ABB RAPID module: Module1.mod

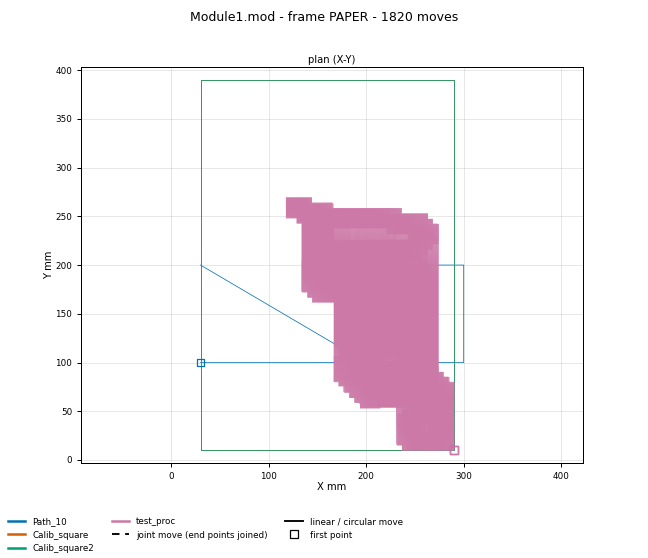
[picture p0: tool path of Module1.mod in frame PAPER, 1820 of 1820 moves have a stored position in this frame; points joined in program order, loops and branches not executed]
MODULE Module1
    CONST robtarget Target_10:=[[30,100,0],[1,0,0,0],[0,0,0,0],[9E+09,9E+09,9E+09,9E+09,9E+09,9E+09]];
    CONST robtarget Target_20:=[[300,100,0],[1,0,0,0],[0,0,0,0],[9E+09,9E+09,9E+09,9E+09,9E+09,9E+09]];
    CONST robtarget Target_30:=[[300,200,0],[1,0,0,0],[0,0,0,0],[9E+09,9E+09,9E+09,9E+09,9E+09,9E+09]];
    CONST robtarget Target_40:=[[200,200,0],[1,0,0,0],[0,0,0,0],[9E+09,9E+09,9E+09,9E+09,9E+09,9E+09]];
    CONST robtarget Target_50:=[[200,100,0],[1,0,0,0],[0,0,0,0],[9E+09,9E+09,9E+09,9E+09,9E+09,9E+09]];
    CONST robtarget Target_60:=[[30,200,0],[1,0,0,0],[0,0,0,0],[9E+09,9E+09,9E+09,9E+09,9E+09,9E+09]];
    CONST robtarget Target_drawing_origin:=[[290,10,-2],[1,0,0,0],[0,0,0,0],[9E+09,9E+09,9E+09,9E+09,9E+09,9E+09]];
!***********************************************************
    !
    ! Module:  Module1
    !
    ! Description:
    !   <Insert description here>
    !
    ! Author: jurdo
    !
    ! Version: 1.0
    !
    !***********************************************************


    !***********************************************************
    !
    ! Procedure main
    !
    !   This is the entry point of your program
    !
    !***********************************************************
    PROC main()

        !Calib_square2;

        test_proc;

    ENDPROC
    PROC Path_10()
        MoveL Target_10,v1000,z0,PencilHolder\WObj:=PAPER;
        MoveL Target_20,v1000,z0,PencilHolder\WObj:=PAPER;
        MoveL Target_30,v1000,z0,PencilHolder\WObj:=PAPER;
        MoveL Target_40,v1000,z0,PencilHolder\WObj:=PAPER;
        MoveL Target_50,v1000,z0,PencilHolder\WObj:=PAPER;
        MoveL Target_60,v1000,z0,PencilHolder\WObj:=PAPER;
    ENDPROC

    PROC Calib_square()
        VAR num width := 380;
        VAR num height := 260;

        MoveJ Offs(Target_drawing_origin,0,0,0),v100,fine,PencilHolder\WObj:=PAPER;

        MoveL Offs(Target_drawing_origin,0,width,0),v100,fine,PencilHolder\WObj:=PAPER;

        MoveL Offs(Target_drawing_origin,-height,width,0),v100,fine,PencilHolder\WObj:=PAPER;

        MoveL Offs(Target_drawing_origin,-height,0,0),v100,fine,PencilHolder\WObj:=PAPER;

        MoveL Offs(Target_drawing_origin,0,0,0),v100,fine,PencilHolder\WObj:=PAPER;

    ENDPROC

    PROC Calib_square2()
    MoveJ Offs(Target_drawing_origin,0,0,0),v100,fine,PencilHolder\WObj:=PAPER;
    MoveL Offs(Target_drawing_origin,0,380,0),v100,fine,PencilHolder\WObj:=PAPER;
    MoveL Offs(Target_drawing_origin,-260,380,0),v100,fine,PencilHolder\WObj:=PAPER;
    MoveL Offs(Target_drawing_origin,-260,0,0),v100,fine,PencilHolder\WObj:=PAPER;
    MoveL Offs(Target_drawing_origin,0,0,0),v100,fine,PencilHolder\WObj:=PAPER;
ENDPROC

! Main procedure
PROC test_proc()


! Draw grey
MoveJ Offs(Target_drawing_origin,0,0,0),v100,fine,PencilHolder\WObj:=PAPER;
MoveL Offs(Target_drawing_origin,0,0,0),v50,fine,PencilHolder\WObj:=PAPER;
MoveL Offs(Target_drawing_origin,0,21,0),v50,fine,PencilHolder\WObj:=PAPER;
MoveL Offs(Target_drawing_origin,0,49,0),v50,fine,PencilHolder\WObj:=PAPER;
MoveL Offs(Target_drawing_origin,0,70,0),v50,fine,PencilHolder\WObj:=PAPER;
MoveL Offs(Target_drawing_origin,-1,0,0),v50,fine,PencilHolder\WObj:=PAPER;
MoveL Offs(Target_drawing_origin,-1,21,0),v50,fine,PencilHolder\WObj:=PAPER;
MoveL Offs(Target_drawing_origin,-1,49,0),v50,fine,PencilHolder\WObj:=PAPER;
MoveL Offs(Target_drawing_origin,-1,70,0),v50,fine,PencilHolder\WObj:=PAPER;
MoveL Offs(Target_drawing_origin,-2,0,0),v50,fine,PencilHolder\WObj:=PAPER;
MoveL Offs(Target_drawing_origin,-2,21,0),v50,fine,PencilHolder\WObj:=PAPER;
MoveL Offs(Target_drawing_origin,-2,49,0),v50,fine,PencilHolder\WObj:=PAPER;
MoveL Offs(Target_drawing_origin,-2,70,0),v50,fine,PencilHolder\WObj:=PAPER;
MoveL Offs(Target_drawing_origin,-3,0,0),v50,fine,PencilHolder\WObj:=PAPER;
MoveL Offs(Target_drawing_origin,-3,21,0),v50,fine,PencilHolder\WObj:=PAPER;
MoveL Offs(Target_drawing_origin,-3,49,0),v50,fine,PencilHolder\WObj:=PAPER;
MoveL Offs(Target_drawing_origin,-3,70,0),v50,fine,PencilHolder\WObj:=PAPER;
MoveL Offs(Target_drawing_origin,-4,0,0),v50,fine,PencilHolder\WObj:=PAPER;
MoveL Offs(Target_drawing_origin,-4,21,0),v50,fine,PencilHolder\WObj:=PAPER;
MoveL Offs(Target_drawing_origin,-4,49,0),v50,fine,PencilHolder\WObj:=PAPER;
MoveL Offs(Target_drawing_origin,-4,70,0),v50,fine,PencilHolder\WObj:=PAPER;
MoveL Offs(Target_drawing_origin,-5,0,0),v50,fine,PencilHolder\WObj:=PAPER;
MoveL Offs(Target_drawing_origin,-5,21,0),v50,fine,PencilHolder\WObj:=PAPER;
MoveL Offs(Target_drawing_origin,-5,44,0),v50,fine,PencilHolder\WObj:=PAPER;
MoveL Offs(Target_drawing_origin,-5,75,0),v50,fine,PencilHolder\WObj:=PAPER;
MoveL Offs(Target_drawing_origin,-6,0,0),v50,fine,PencilHolder\WObj:=PAPER;
MoveL Offs(Target_drawing_origin,-6,21,0),v50,fine,PencilHolder\WObj:=PAPER;
MoveL Offs(Target_drawing_origin,-6,43,0),v50,fine,PencilHolder\WObj:=PAPER;
MoveL Offs(Target_drawing_origin,-6,75,0),v50,fine,PencilHolder\WObj:=PAPER;
MoveL Offs(Target_drawing_origin,-7,0,0),v50,fine,PencilHolder\WObj:=PAPER;
MoveL Offs(Target_drawing_origin,-7,21,0),v50,fine,PencilHolder\WObj:=PAPER;
MoveL Offs(Target_drawing_origin,-7,43,0),v50,fine,PencilHolder\WObj:=PAPER;
MoveL Offs(Target_drawing_origin,-7,75,0),v50,fine,PencilHolder\WObj:=PAPER;
MoveL Offs(Target_drawing_origin,-8,0,0),v50,fine,PencilHolder\WObj:=PAPER;
MoveL Offs(Target_drawing_origin,-8,21,0),v50,fine,PencilHolder\WObj:=PAPER;
MoveL Offs(Target_drawing_origin,-8,43,0),v50,fine,PencilHolder\WObj:=PAPER;
MoveL Offs(Target_drawing_origin,-8,75,0),v50,fine,PencilHolder\WObj:=PAPER;
MoveL Offs(Target_drawing_origin,-9,0,0),v50,fine,PencilHolder\WObj:=PAPER;
MoveL Offs(Target_drawing_origin,-9,21,0),v50,fine,PencilHolder\WObj:=PAPER;
MoveL Offs(Target_drawing_origin,-9,43,0),v50,fine,PencilHolder\WObj:=PAPER;
MoveL Offs(Target_drawing_origin,-9,75,0),v50,fine,PencilHolder\WObj:=PAPER;
MoveL Offs(Target_drawing_origin,-10,0,0),v50,fine,PencilHolder\WObj:=PAPER;
MoveL Offs(Target_drawing_origin,-10,21,0),v50,fine,PencilHolder\WObj:=PAPER;
MoveL Offs(Target_drawing_origin,-10,43,0),v50,fine,PencilHolder\WObj:=PAPER;
MoveL Offs(Target_drawing_origin,-10,75,0),v50,fine,PencilHolder\WObj:=PAPER;
MoveL Offs(Target_drawing_origin,-11,0,0),v50,fine,PencilHolder\WObj:=PAPER;
MoveL Offs(Target_drawing_origin,-11,21,0),v50,fine,PencilHolder\WObj:=PAPER;
MoveL Offs(Target_drawing_origin,-11,38,0),v50,fine,PencilHolder\WObj:=PAPER;
MoveL Offs(Target_drawing_origin,-11,80,0),v50,fine,PencilHolder\WObj:=PAPER;
MoveL Offs(Target_drawing_origin,-12,0,0),v50,fine,PencilHolder\WObj:=PAPER;
MoveL Offs(Target_drawing_origin,-12,21,0),v50,fine,PencilHolder\WObj:=PAPER;
MoveL Offs(Target_drawing_origin,-12,38,0),v50,fine,PencilHolder\WObj:=PAPER;
MoveL Offs(Target_drawing_origin,-12,80,0),v50,fine,PencilHolder\WObj:=PAPER;
MoveL Offs(Target_drawing_origin,-13,0,0),v50,fine,PencilHolder\WObj:=PAPER;
MoveL Offs(Target_drawing_origin,-13,21,0),v50,fine,PencilHolder\WObj:=PAPER;
MoveL Offs(Target_drawing_origin,-13,38,0),v50,fine,PencilHolder\WObj:=PAPER;
MoveL Offs(Target_drawing_origin,-13,80,0),v50,fine,PencilHolder\WObj:=PAPER;
MoveL Offs(Target_drawing_origin,-14,0,0),v50,fine,PencilHolder\WObj:=PAPER;
MoveL Offs(Target_drawing_origin,-14,21,0),v50,fine,PencilHolder\WObj:=PAPER;
MoveL Offs(Target_drawing_origin,-14,38,0),v50,fine,PencilHolder\WObj:=PAPER;
MoveL Offs(Target_drawing_origin,-14,80,0),v50,fine,PencilHolder\WObj:=PAPER;
MoveL Offs(Target_drawing_origin,-15,0,0),v50,fine,PencilHolder\WObj:=PAPER;
MoveL Offs(Target_drawing_origin,-15,21,0),v50,fine,PencilHolder\WObj:=PAPER;
MoveL Offs(Target_drawing_origin,-15,38,0),v50,fine,PencilHolder\WObj:=PAPER;
MoveL Offs(Target_drawing_origin,-15,80,0),v50,fine,PencilHolder\WObj:=PAPER;
MoveL Offs(Target_drawing_origin,-16,0,0),v50,fine,PencilHolder\WObj:=PAPER;
MoveL Offs(Target_drawing_origin,-16,16,0),v50,fine,PencilHolder\WObj:=PAPER;
MoveL Offs(Target_drawing_origin,-16,27,0),v50,fine,PencilHolder\WObj:=PAPER;
MoveL Offs(Target_drawing_origin,-16,86,0),v50,fine,PencilHolder\WObj:=PAPER;
MoveL Offs(Target_drawing_origin,-16,211,0),v50,fine,PencilHolder\WObj:=PAPER;
MoveL Offs(Target_drawing_origin,-16,232,0),v50,fine,PencilHolder\WObj:=PAPER;
MoveL Offs(Target_drawing_origin,-17,0,0),v50,fine,PencilHolder\WObj:=PAPER;
MoveL Offs(Target_drawing_origin,-17,15,0),v50,fine,PencilHolder\WObj:=PAPER;
MoveL Offs(Target_drawing_origin,-17,27,0),v50,fine,PencilHolder\WObj:=PAPER;
MoveL Offs(Target_drawing_origin,-17,86,0),v50,fine,PencilHolder\WObj:=PAPER;
MoveL Offs(Target_drawing_origin,-17,211,0),v50,fine,PencilHolder\WObj:=PAPER;
MoveL Offs(Target_drawing_origin,-17,232,0),v50,fine,PencilHolder\WObj:=PAPER;
MoveL Offs(Target_drawing_origin,-18,0,0),v50,fine,PencilHolder\WObj:=PAPER;
MoveL Offs(Target_drawing_origin,-18,15,0),v50,fine,PencilHolder\WObj:=PAPER;
MoveL Offs(Target_drawing_origin,-18,27,0),v50,fine,PencilHolder\WObj:=PAPER;
MoveL Offs(Target_drawing_origin,-18,86,0),v50,fine,PencilHolder\WObj:=PAPER;
MoveL Offs(Target_drawing_origin,-18,211,0),v50,fine,PencilHolder\WObj:=PAPER;
MoveL Offs(Target_drawing_origin,-18,232,0),v50,fine,PencilHolder\WObj:=PAPER;
MoveL Offs(Target_drawing_origin,-19,0,0),v50,fine,PencilHolder\WObj:=PAPER;
MoveL Offs(Target_drawing_origin,-19,15,0),v50,fine,PencilHolder\WObj:=PAPER;
MoveL Offs(Target_drawing_origin,-19,27,0),v50,fine,PencilHolder\WObj:=PAPER;
MoveL Offs(Target_drawing_origin,-19,86,0),v50,fine,PencilHolder\WObj:=PAPER;
MoveL Offs(Target_drawing_origin,-19,211,0),v50,fine,PencilHolder\WObj:=PAPER;
MoveL Offs(Target_drawing_origin,-19,232,0),v50,fine,PencilHolder\WObj:=PAPER;
MoveL Offs(Target_drawing_origin,-20,0,0),v50,fine,PencilHolder\WObj:=PAPER;
MoveL Offs(Target_drawing_origin,-20,15,0),v50,fine,PencilHolder\WObj:=PAPER;
MoveL Offs(Target_drawing_origin,-20,27,0),v50,fine,PencilHolder\WObj:=PAPER;
MoveL Offs(Target_drawing_origin,-20,86,0),v50,fine,PencilHolder\WObj:=PAPER;
MoveL Offs(Target_drawing_origin,-20,211,0),v50,fine,PencilHolder\WObj:=PAPER;
MoveL Offs(Target_drawing_origin,-20,232,0),v50,fine,PencilHolder\WObj:=PAPER;
MoveL Offs(Target_drawing_origin,-21,0,0),v50,fine,PencilHolder\WObj:=PAPER;
MoveL Offs(Target_drawing_origin,-21,15,0),v50,fine,PencilHolder\WObj:=PAPER;
MoveL Offs(Target_drawing_origin,-21,27,0),v50,fine,PencilHolder\WObj:=PAPER;
MoveL Offs(Target_drawing_origin,-21,86,0),v50,fine,PencilHolder\WObj:=PAPER;
MoveL Offs(Target_drawing_origin,-21,211,0),v50,fine,PencilHolder\WObj:=PAPER;
MoveL Offs(Target_drawing_origin,-21,232,0),v50,fine,PencilHolder\WObj:=PAPER;
MoveL Offs(Target_drawing_origin,-22,0,0),v50,fine,PencilHolder\WObj:=PAPER;
MoveL Offs(Target_drawing_origin,-22,15,0),v50,fine,PencilHolder\WObj:=PAPER;
MoveL Offs(Target_drawing_origin,-22,27,0),v50,fine,PencilHolder\WObj:=PAPER;
MoveL Offs(Target_drawing_origin,-22,91,0),v50,fine,PencilHolder\WObj:=PAPER;
MoveL Offs(Target_drawing_origin,-22,206,0),v50,fine,PencilHolder\WObj:=PAPER;
MoveL Offs(Target_drawing_origin,-22,237,0),v50,fine,PencilHolder\WObj:=PAPER;
MoveL Offs(Target_drawing_origin,-23,0,0),v50,fine,PencilHolder\WObj:=PAPER;
MoveL Offs(Target_drawing_origin,-23,15,0),v50,fine,PencilHolder\WObj:=PAPER;
MoveL Offs(Target_drawing_origin,-23,27,0),v50,fine,PencilHolder\WObj:=PAPER;
MoveL Offs(Target_drawing_origin,-23,91,0),v50,fine,PencilHolder\WObj:=PAPER;
MoveL Offs(Target_drawing_origin,-23,206,0),v50,fine,PencilHolder\WObj:=PAPER;
MoveL Offs(Target_drawing_origin,-23,237,0),v50,fine,PencilHolder\WObj:=PAPER;
MoveL Offs(Target_drawing_origin,-24,0,0),v50,fine,PencilHolder\WObj:=PAPER;
MoveL Offs(Target_drawing_origin,-24,15,0),v50,fine,PencilHolder\WObj:=PAPER;
MoveL Offs(Target_drawing_origin,-24,27,0),v50,fine,PencilHolder\WObj:=PAPER;
MoveL Offs(Target_drawing_origin,-24,91,0),v50,fine,PencilHolder\WObj:=PAPER;
MoveL Offs(Target_drawing_origin,-24,206,0),v50,fine,PencilHolder\WObj:=PAPER;
MoveL Offs(Target_drawing_origin,-24,237,0),v50,fine,PencilHolder\WObj:=PAPER;
MoveL Offs(Target_drawing_origin,-25,0,0),v50,fine,PencilHolder\WObj:=PAPER;
MoveL Offs(Target_drawing_origin,-25,15,0),v50,fine,PencilHolder\WObj:=PAPER;
MoveL Offs(Target_drawing_origin,-25,27,0),v50,fine,PencilHolder\WObj:=PAPER;
MoveL Offs(Target_drawing_origin,-25,91,0),v50,fine,PencilHolder\WObj:=PAPER;
MoveL Offs(Target_drawing_origin,-25,206,0),v50,fine,PencilHolder\WObj:=PAPER;
MoveL Offs(Target_drawing_origin,-25,237,0),v50,fine,PencilHolder\WObj:=PAPER;
MoveL Offs(Target_drawing_origin,-26,0,0),v50,fine,PencilHolder\WObj:=PAPER;
MoveL Offs(Target_drawing_origin,-26,15,0),v50,fine,PencilHolder\WObj:=PAPER;
MoveL Offs(Target_drawing_origin,-26,27,0),v50,fine,PencilHolder\WObj:=PAPER;
MoveL Offs(Target_drawing_origin,-26,91,0),v50,fine,PencilHolder\WObj:=PAPER;
MoveL Offs(Target_drawing_origin,-26,206,0),v50,fine,PencilHolder\WObj:=PAPER;
MoveL Offs(Target_drawing_origin,-26,237,0),v50,fine,PencilHolder\WObj:=PAPER;
MoveL Offs(Target_drawing_origin,-27,0,0),v50,fine,PencilHolder\WObj:=PAPER;
MoveL Offs(Target_drawing_origin,-27,91,0),v50,fine,PencilHolder\WObj:=PAPER;
MoveL Offs(Target_drawing_origin,-27,131,0),v50,fine,PencilHolder\WObj:=PAPER;
MoveL Offs(Target_drawing_origin,-27,156,0),v50,fine,PencilHolder\WObj:=PAPER;
MoveL Offs(Target_drawing_origin,-27,200,0),v50,fine,PencilHolder\WObj:=PAPER;
MoveL Offs(Target_drawing_origin,-27,243,0),v50,fine,PencilHolder\WObj:=PAPER;
MoveL Offs(Target_drawing_origin,-28,0,0),v50,fine,PencilHolder\WObj:=PAPER;
MoveL Offs(Target_drawing_origin,-28,91,0),v50,fine,PencilHolder\WObj:=PAPER;
MoveL Offs(Target_drawing_origin,-28,131,0),v50,fine,PencilHolder\WObj:=PAPER;
MoveL Offs(Target_drawing_origin,-28,156,0),v50,fine,PencilHolder\WObj:=PAPER;
MoveL Offs(Target_drawing_origin,-28,200,0),v50,fine,PencilHolder\WObj:=PAPER;
MoveL Offs(Target_drawing_origin,-28,243,0),v50,fine,PencilHolder\WObj:=PAPER;
MoveL Offs(Target_drawing_origin,-29,0,0),v50,fine,PencilHolder\WObj:=PAPER;
MoveL Offs(Target_drawing_origin,-29,91,0),v50,fine,PencilHolder\WObj:=PAPER;
MoveL Offs(Target_drawing_origin,-29,131,0),v50,fine,PencilHolder\WObj:=PAPER;
MoveL Offs(Target_drawing_origin,-29,156,0),v50,fine,PencilHolder\WObj:=PAPER;
MoveL Offs(Target_drawing_origin,-29,200,0),v50,fine,PencilHolder\WObj:=PAPER;
MoveL Offs(Target_drawing_origin,-29,243,0),v50,fine,PencilHolder\WObj:=PAPER;
MoveL Offs(Target_drawing_origin,-30,0,0),v50,fine,PencilHolder\WObj:=PAPER;
MoveL Offs(Target_drawing_origin,-30,91,0),v50,fine,PencilHolder\WObj:=PAPER;
MoveL Offs(Target_drawing_origin,-30,131,0),v50,fine,PencilHolder\WObj:=PAPER;
MoveL Offs(Target_drawing_origin,-30,156,0),v50,fine,PencilHolder\WObj:=PAPER;
MoveL Offs(Target_drawing_origin,-30,200,0),v50,fine,PencilHolder\WObj:=PAPER;
MoveL Offs(Target_drawing_origin,-30,243,0),v50,fine,PencilHolder\WObj:=PAPER;
MoveL Offs(Target_drawing_origin,-31,0,0),v50,fine,PencilHolder\WObj:=PAPER;
MoveL Offs(Target_drawing_origin,-31,91,0),v50,fine,PencilHolder\WObj:=PAPER;
MoveL Offs(Target_drawing_origin,-31,131,0),v50,fine,PencilHolder\WObj:=PAPER;
MoveL Offs(Target_drawing_origin,-31,156,0),v50,fine,PencilHolder\WObj:=PAPER;
MoveL Offs(Target_drawing_origin,-31,200,0),v50,fine,PencilHolder\WObj:=PAPER;
MoveL Offs(Target_drawing_origin,-31,243,0),v50,fine,PencilHolder\WObj:=PAPER;
MoveL Offs(Target_drawing_origin,-32,0,0),v50,fine,PencilHolder\WObj:=PAPER;
MoveL Offs(Target_drawing_origin,-32,91,0),v50,fine,PencilHolder\WObj:=PAPER;
MoveL Offs(Target_drawing_origin,-32,125,0),v50,fine,PencilHolder\WObj:=PAPER;
MoveL Offs(Target_drawing_origin,-32,161,0),v50,fine,PencilHolder\WObj:=PAPER;
MoveL Offs(Target_drawing_origin,-32,195,0),v50,fine,PencilHolder\WObj:=PAPER;
MoveL Offs(Target_drawing_origin,-32,243,0),v50,fine,PencilHolder\WObj:=PAPER;
MoveL Offs(Target_drawing_origin,-33,0,0),v50,fine,PencilHolder\WObj:=PAPER;
MoveL Offs(Target_drawing_origin,-33,53,0),v50,fine,PencilHolder\WObj:=PAPER;
MoveL Offs(Target_drawing_origin,-33,59,0),v50,fine,PencilHolder\WObj:=PAPER;
MoveL Offs(Target_drawing_origin,-33,91,0),v50,fine,PencilHolder\WObj:=PAPER;
MoveL Offs(Target_drawing_origin,-33,124,0),v50,fine,PencilHolder\WObj:=PAPER;
MoveL Offs(Target_drawing_origin,-33,162,0),v50,fine,PencilHolder\WObj:=PAPER;
MoveL Offs(Target_drawing_origin,-33,195,0),v50,fine,PencilHolder\WObj:=PAPER;
MoveL Offs(Target_drawing_origin,-33,243,0),v50,fine,PencilHolder\WObj:=PAPER;
MoveL Offs(Target_drawing_origin,-34,0,0),v50,fine,PencilHolder\WObj:=PAPER;
MoveL Offs(Target_drawing_origin,-34,53,0),v50,fine,PencilHolder\WObj:=PAPER;
MoveL Offs(Target_drawing_origin,-34,59,0),v50,fine,PencilHolder\WObj:=PAPER;
MoveL Offs(Target_drawing_origin,-34,91,0),v50,fine,PencilHolder\WObj:=PAPER;
MoveL Offs(Target_drawing_origin,-34,124,0),v50,fine,PencilHolder\WObj:=PAPER;
MoveL Offs(Target_drawing_origin,-34,162,0),v50,fine,PencilHolder\WObj:=PAPER;
MoveL Offs(Target_drawing_origin,-34,195,0),v50,fine,PencilHolder\WObj:=PAPER;
MoveL Offs(Target_drawing_origin,-34,243,0),v50,fine,PencilHolder\WObj:=PAPER;
MoveL Offs(Target_drawing_origin,-35,0,0),v50,fine,PencilHolder\WObj:=PAPER;
MoveL Offs(Target_drawing_origin,-35,53,0),v50,fine,PencilHolder\WObj:=PAPER;
MoveL Offs(Target_drawing_origin,-35,59,0),v50,fine,PencilHolder\WObj:=PAPER;
MoveL Offs(Target_drawing_origin,-35,91,0),v50,fine,PencilHolder\WObj:=PAPER;
MoveL Offs(Target_drawing_origin,-35,124,0),v50,fine,PencilHolder\WObj:=PAPER;
MoveL Offs(Target_drawing_origin,-35,162,0),v50,fine,PencilHolder\WObj:=PAPER;
MoveL Offs(Target_drawing_origin,-35,195,0),v50,fine,PencilHolder\WObj:=PAPER;
MoveL Offs(Target_drawing_origin,-35,243,0),v50,fine,PencilHolder\WObj:=PAPER;
MoveL Offs(Target_drawing_origin,-36,0,0),v50,fine,PencilHolder\WObj:=PAPER;
MoveL Offs(Target_drawing_origin,-36,53,0),v50,fine,PencilHolder\WObj:=PAPER;
MoveL Offs(Target_drawing_origin,-36,59,0),v50,fine,PencilHolder\WObj:=PAPER;
MoveL Offs(Target_drawing_origin,-36,91,0),v50,fine,PencilHolder\WObj:=PAPER;
MoveL Offs(Target_drawing_origin,-36,124,0),v50,fine,PencilHolder\WObj:=PAPER;
MoveL Offs(Target_drawing_origin,-36,162,0),v50,fine,PencilHolder\WObj:=PAPER;
MoveL Offs(Target_drawing_origin,-36,195,0),v50,fine,PencilHolder\WObj:=PAPER;
MoveL Offs(Target_drawing_origin,-36,243,0),v50,fine,PencilHolder\WObj:=PAPER;
MoveL Offs(Target_drawing_origin,-37,0,0),v50,fine,PencilHolder\WObj:=PAPER;
MoveL Offs(Target_drawing_origin,-37,53,0),v50,fine,PencilHolder\WObj:=PAPER;
MoveL Offs(Target_drawing_origin,-37,59,0),v50,fine,PencilHolder\WObj:=PAPER;
MoveL Offs(Target_drawing_origin,-37,91,0),v50,fine,PencilHolder\WObj:=PAPER;
MoveL Offs(Target_drawing_origin,-37,124,0),v50,fine,PencilHolder\WObj:=PAPER;
MoveL Offs(Target_drawing_origin,-37,162,0),v50,fine,PencilHolder\WObj:=PAPER;
MoveL Offs(Target_drawing_origin,-37,195,0),v50,fine,PencilHolder\WObj:=PAPER;
MoveL Offs(Target_drawing_origin,-37,243,0),v50,fine,PencilHolder\WObj:=PAPER;
MoveL Offs(Target_drawing_origin,-38,0,0),v50,fine,PencilHolder\WObj:=PAPER;
MoveL Offs(Target_drawing_origin,-38,48,0),v50,fine,PencilHolder\WObj:=PAPER;
MoveL Offs(Target_drawing_origin,-38,59,0),v50,fine,PencilHolder\WObj:=PAPER;
MoveL Offs(Target_drawing_origin,-38,91,0),v50,fine,PencilHolder\WObj:=PAPER;
MoveL Offs(Target_drawing_origin,-38,114,0),v50,fine,PencilHolder\WObj:=PAPER;
MoveL Offs(Target_drawing_origin,-38,167,0),v50,fine,PencilHolder\WObj:=PAPER;
MoveL Offs(Target_drawing_origin,-38,195,0),v50,fine,PencilHolder\WObj:=PAPER;
MoveL Offs(Target_drawing_origin,-38,243,0),v50,fine,PencilHolder\WObj:=PAPER;
MoveL Offs(Target_drawing_origin,-39,0,0),v50,fine,PencilHolder\WObj:=PAPER;
MoveL Offs(Target_drawing_origin,-39,48,0),v50,fine,PencilHolder\WObj:=PAPER;
MoveL Offs(Target_drawing_origin,-39,59,0),v50,fine,PencilHolder\WObj:=PAPER;
MoveL Offs(Target_drawing_origin,-39,91,0),v50,fine,PencilHolder\WObj:=PAPER;
MoveL Offs(Target_drawing_origin,-39,114,0),v50,fine,PencilHolder\WObj:=PAPER;
MoveL Offs(Target_drawing_origin,-39,167,0),v50,fine,PencilHolder\WObj:=PAPER;
MoveL Offs(Target_drawing_origin,-39,195,0),v50,fine,PencilHolder\WObj:=PAPER;
MoveL Offs(Target_drawing_origin,-39,243,0),v50,fine,PencilHolder\WObj:=PAPER;
MoveL Offs(Target_drawing_origin,-40,0,0),v50,fine,PencilHolder\WObj:=PAPER;
MoveL Offs(Target_drawing_origin,-40,48,0),v50,fine,PencilHolder\WObj:=PAPER;
MoveL Offs(Target_drawing_origin,-40,59,0),v50,fine,PencilHolder\WObj:=PAPER;
MoveL Offs(Target_drawing_origin,-40,91,0),v50,fine,PencilHolder\WObj:=PAPER;
MoveL Offs(Target_drawing_origin,-40,114,0),v50,fine,PencilHolder\WObj:=PAPER;
MoveL Offs(Target_drawing_origin,-40,167,0),v50,fine,PencilHolder\WObj:=PAPER;
MoveL Offs(Target_drawing_origin,-40,195,0),v50,fine,PencilHolder\WObj:=PAPER;
MoveL Offs(Target_drawing_origin,-40,243,0),v50,fine,PencilHolder\WObj:=PAPER;
MoveL Offs(Target_drawing_origin,-41,0,0),v50,fine,PencilHolder\WObj:=PAPER;
MoveL Offs(Target_drawing_origin,-41,48,0),v50,fine,PencilHolder\WObj:=PAPER;
MoveL Offs(Target_drawing_origin,-41,59,0),v50,fine,PencilHolder\WObj:=PAPER;
MoveL Offs(Target_drawing_origin,-41,91,0),v50,fine,PencilHolder\WObj:=PAPER;
MoveL Offs(Target_drawing_origin,-41,114,0),v50,fine,PencilHolder\WObj:=PAPER;
MoveL Offs(Target_drawing_origin,-41,167,0),v50,fine,PencilHolder\WObj:=PAPER;
MoveL Offs(Target_drawing_origin,-41,195,0),v50,fine,PencilHolder\WObj:=PAPER;
MoveL Offs(Target_drawing_origin,-41,243,0),v50,fine,PencilHolder\WObj:=PAPER;
MoveL Offs(Target_drawing_origin,-42,0,0),v50,fine,PencilHolder\WObj:=PAPER;
MoveL Offs(Target_drawing_origin,-42,48,0),v50,fine,PencilHolder\WObj:=PAPER;
MoveL Offs(Target_drawing_origin,-42,59,0),v50,fine,PencilHolder\WObj:=PAPER;
MoveL Offs(Target_drawing_origin,-42,91,0),v50,fine,PencilHolder\WObj:=PAPER;
MoveL Offs(Target_drawing_origin,-42,114,0),v50,fine,PencilHolder\WObj:=PAPER;
MoveL Offs(Target_drawing_origin,-42,167,0),v50,fine,PencilHolder\WObj:=PAPER;
MoveL Offs(Target_drawing_origin,-42,195,0),v50,fine,PencilHolder\WObj:=PAPER;
MoveL Offs(Target_drawing_origin,-42,243,0),v50,fine,PencilHolder\WObj:=PAPER;
MoveL Offs(Target_drawing_origin,-43,0,0),v50,fine,PencilHolder\WObj:=PAPER;
MoveL Offs(Target_drawing_origin,-43,43,0),v50,fine,PencilHolder\WObj:=PAPER;
MoveL Offs(Target_drawing_origin,-43,59,0),v50,fine,PencilHolder\WObj:=PAPER;
MoveL Offs(Target_drawing_origin,-43,91,0),v50,fine,PencilHolder\WObj:=PAPER;
MoveL Offs(Target_drawing_origin,-43,108,0),v50,fine,PencilHolder\WObj:=PAPER;
MoveL Offs(Target_drawing_origin,-43,172,0),v50,fine,PencilHolder\WObj:=PAPER;
MoveL Offs(Target_drawing_origin,-43,190,0),v50,fine,PencilHolder\WObj:=PAPER;
MoveL Offs(Target_drawing_origin,-43,243,0),v50,fine,PencilHolder\WObj:=PAPER;
MoveL Offs(Target_drawing_origin,-44,0,0),v50,fine,PencilHolder\WObj:=PAPER;
MoveL Offs(Target_drawing_origin,-44,42,0),v50,fine,PencilHolder\WObj:=PAPER;
MoveL Offs(Target_drawing_origin,-44,59,0),v50,fine,PencilHolder\WObj:=PAPER;
MoveL Offs(Target_drawing_origin,-44,91,0),v50,fine,PencilHolder\WObj:=PAPER;
MoveL Offs(Target_drawing_origin,-44,108,0),v50,fine,PencilHolder\WObj:=PAPER;
MoveL Offs(Target_drawing_origin,-44,172,0),v50,fine,PencilHolder\WObj:=PAPER;
MoveL Offs(Target_drawing_origin,-44,189,0),v50,fine,PencilHolder\WObj:=PAPER;
MoveL Offs(Target_drawing_origin,-44,243,0),v50,fine,PencilHolder\WObj:=PAPER;
MoveL Offs(Target_drawing_origin,-45,0,0),v50,fine,PencilHolder\WObj:=PAPER;
MoveL Offs(Target_drawing_origin,-45,42,0),v50,fine,PencilHolder\WObj:=PAPER;
MoveL Offs(Target_drawing_origin,-45,59,0),v50,fine,PencilHolder\WObj:=PAPER;
MoveL Offs(Target_drawing_origin,-45,91,0),v50,fine,PencilHolder\WObj:=PAPER;
MoveL Offs(Target_drawing_origin,-45,108,0),v50,fine,PencilHolder\WObj:=PAPER;
MoveL Offs(Target_drawing_origin,-45,172,0),v50,fine,PencilHolder\WObj:=PAPER;
MoveL Offs(Target_drawing_origin,-45,189,0),v50,fine,PencilHolder\WObj:=PAPER;
MoveL Offs(Target_drawing_origin,-45,243,0),v50,fine,PencilHolder\WObj:=PAPER;
MoveL Offs(Target_drawing_origin,-46,0,0),v50,fine,PencilHolder\WObj:=PAPER;
MoveL Offs(Target_drawing_origin,-46,42,0),v50,fine,PencilHolder\WObj:=PAPER;
MoveL Offs(Target_drawing_origin,-46,59,0),v50,fine,PencilHolder\WObj:=PAPER;
MoveL Offs(Target_drawing_origin,-46,91,0),v50,fine,PencilHolder\WObj:=PAPER;
MoveL Offs(Target_drawing_origin,-46,108,0),v50,fine,PencilHolder\WObj:=PAPER;
MoveL Offs(Target_drawing_origin,-46,172,0),v50,fine,PencilHolder\WObj:=PAPER;
MoveL Offs(Target_drawing_origin,-46,189,0),v50,fine,PencilHolder\WObj:=PAPER;
MoveL Offs(Target_drawing_origin,-46,243,0),v50,fine,PencilHolder\WObj:=PAPER;
MoveL Offs(Target_drawing_origin,-47,0,0),v50,fine,PencilHolder\WObj:=PAPER;
MoveL Offs(Target_drawing_origin,-47,42,0),v50,fine,PencilHolder\WObj:=PAPER;
MoveL Offs(Target_drawing_origin,-47,59,0),v50,fine,PencilHolder\WObj:=PAPER;
MoveL Offs(Target_drawing_origin,-47,91,0),v50,fine,PencilHolder\WObj:=PAPER;
MoveL Offs(Target_drawing_origin,-47,108,0),v50,fine,PencilHolder\WObj:=PAPER;
MoveL Offs(Target_drawing_origin,-47,172,0),v50,fine,PencilHolder\WObj:=PAPER;
MoveL Offs(Target_drawing_origin,-47,189,0),v50,fine,PencilHolder\WObj:=PAPER;
MoveL Offs(Target_drawing_origin,-47,243,0),v50,fine,PencilHolder\WObj:=PAPER;
MoveL Offs(Target_drawing_origin,-48,0,0),v50,fine,PencilHolder\WObj:=PAPER;
MoveL Offs(Target_drawing_origin,-48,42,0),v50,fine,PencilHolder\WObj:=PAPER;
MoveL Offs(Target_drawing_origin,-48,59,0),v50,fine,PencilHolder\WObj:=PAPER;
MoveL Offs(Target_drawing_origin,-48,91,0),v50,fine,PencilHolder\WObj:=PAPER;
MoveL Offs(Target_drawing_origin,-48,108,0),v50,fine,PencilHolder\WObj:=PAPER;
MoveL Offs(Target_drawing_origin,-48,172,0),v50,fine,PencilHolder\WObj:=PAPER;
MoveL Offs(Target_drawing_origin,-48,189,0),v50,fine,PencilHolder\WObj:=PAPER;
MoveL Offs(Target_drawing_origin,-48,243,0),v50,fine,PencilHolder\WObj:=PAPER;
MoveL Offs(Target_drawing_origin,-49,0,0),v50,fine,PencilHolder\WObj:=PAPER;
MoveL Offs(Target_drawing_origin,-49,42,0),v50,fine,PencilHolder\WObj:=PAPER;
MoveL Offs(Target_drawing_origin,-49,59,0),v50,fine,PencilHolder\WObj:=PAPER;
MoveL Offs(Target_drawing_origin,-49,91,0),v50,fine,PencilHolder\WObj:=PAPER;
MoveL Offs(Target_drawing_origin,-49,103,0),v50,fine,PencilHolder\WObj:=PAPER;
MoveL Offs(Target_drawing_origin,-49,172,0),v50,fine,PencilHolder\WObj:=PAPER;
MoveL Offs(Target_drawing_origin,-49,189,0),v50,fine,PencilHolder\WObj:=PAPER;
MoveL Offs(Target_drawing_origin,-49,216,0),v50,fine,PencilHolder\WObj:=PAPER;
MoveL Offs(Target_drawing_origin,-49,222,0),v50,fine,PencilHolder\WObj:=PAPER;
MoveL Offs(Target_drawing_origin,-49,243,0),v50,fine,PencilHolder\WObj:=PAPER;
MoveL Offs(Target_drawing_origin,-50,0,0),v50,fine,PencilHolder\WObj:=PAPER;
MoveL Offs(Target_drawing_origin,-50,42,0),v50,fine,PencilHolder\WObj:=PAPER;
MoveL Offs(Target_drawing_origin,-50,59,0),v50,fine,PencilHolder\WObj:=PAPER;
MoveL Offs(Target_drawing_origin,-50,91,0),v50,fine,PencilHolder\WObj:=PAPER;
MoveL Offs(Target_drawing_origin,-50,103,0),v50,fine,PencilHolder\WObj:=PAPER;
MoveL Offs(Target_drawing_origin,-50,172,0),v50,fine,PencilHolder\WObj:=PAPER;
MoveL Offs(Target_drawing_origin,-50,189,0),v50,fine,PencilHolder\WObj:=PAPER;
MoveL Offs(Target_drawing_origin,-50,216,0),v50,fine,PencilHolder\WObj:=PAPER;
MoveL Offs(Target_drawing_origin,-50,222,0),v50,fine,PencilHolder\WObj:=PAPER;
MoveL Offs(Target_drawing_origin,-50,243,0),v50,fine,PencilHolder\WObj:=PAPER;
MoveL Offs(Target_drawing_origin,-51,0,0),v50,fine,PencilHolder\WObj:=PAPER;
MoveL Offs(Target_drawing_origin,-51,42,0),v50,fine,PencilHolder\WObj:=PAPER;
MoveL Offs(Target_drawing_origin,-51,59,0),v50,fine,PencilHolder\WObj:=PAPER;
MoveL Offs(Target_drawing_origin,-51,91,0),v50,fine,PencilHolder\WObj:=PAPER;
MoveL Offs(Target_drawing_origin,-51,103,0),v50,fine,PencilHolder\WObj:=PAPER;
MoveL Offs(Target_drawing_origin,-51,172,0),v50,fine,PencilHolder\WObj:=PAPER;
MoveL Offs(Target_drawing_origin,-51,189,0),v50,fine,PencilHolder\WObj:=PAPER;
MoveL Offs(Target_drawing_origin,-51,216,0),v50,fine,PencilHolder\WObj:=PAPER;
MoveL Offs(Target_drawing_origin,-51,222,0),v50,fine,PencilHolder\WObj:=PAPER;
MoveL Offs(Target_drawing_origin,-51,243,0),v50,fine,PencilHolder\WObj:=PAPER;
MoveL Offs(Target_drawing_origin,-52,0,0),v50,fine,PencilHolder\WObj:=PAPER;
MoveL Offs(Target_drawing_origin,-52,42,0),v50,fine,PencilHolder\WObj:=PAPER;
MoveL Offs(Target_drawing_origin,-52,59,0),v50,fine,PencilHolder\WObj:=PAPER;
MoveL Offs(Target_drawing_origin,-52,91,0),v50,fine,PencilHolder\WObj:=PAPER;
MoveL Offs(Target_drawing_origin,-52,103,0),v50,fine,PencilHolder\WObj:=PAPER;
MoveL Offs(Target_drawing_origin,-52,172,0),v50,fine,PencilHolder\WObj:=PAPER;
MoveL Offs(Target_drawing_origin,-52,189,0),v50,fine,PencilHolder\WObj:=PAPER;
MoveL Offs(Target_drawing_origin,-52,216,0),v50,fine,PencilHolder\WObj:=PAPER;
MoveL Offs(Target_drawing_origin,-52,222,0),v50,fine,PencilHolder\WObj:=PAPER;
MoveL Offs(Target_drawing_origin,-52,243,0),v50,fine,PencilHolder\WObj:=PAPER;
MoveL Offs(Target_drawing_origin,-53,0,0),v50,fine,PencilHolder\WObj:=PAPER;
MoveL Offs(Target_drawing_origin,-53,42,0),v50,fine,PencilHolder\WObj:=PAPER;
MoveL Offs(Target_drawing_origin,-53,59,0),v50,fine,PencilHolder\WObj:=PAPER;
MoveL Offs(Target_drawing_origin,-53,91,0),v50,fine,PencilHolder\WObj:=PAPER;
MoveL Offs(Target_drawing_origin,-53,103,0),v50,fine,PencilHolder\WObj:=PAPER;
MoveL Offs(Target_drawing_origin,-53,172,0),v50,fine,PencilHolder\WObj:=PAPER;
MoveL Offs(Target_drawing_origin,-53,189,0),v50,fine,PencilHolder\WObj:=PAPER;
MoveL Offs(Target_drawing_origin,-53,216,0),v50,fine,PencilHolder\WObj:=PAPER;
MoveL Offs(Target_drawing_origin,-53,222,0),v50,fine,PencilHolder\WObj:=PAPER;
MoveL Offs(Target_drawing_origin,-53,243,0),v50,fine,PencilHolder\WObj:=PAPER;
MoveL Offs(Target_drawing_origin,-54,5,0),v50,fine,PencilHolder\WObj:=PAPER;
MoveL Offs(Target_drawing_origin,-54,37,0),v50,fine,PencilHolder\WObj:=PAPER;
MoveL Offs(Target_drawing_origin,-54,59,0),v50,fine,PencilHolder\WObj:=PAPER;
MoveL Offs(Target_drawing_origin,-54,91,0),v50,fine,PencilHolder\WObj:=PAPER;
MoveL Offs(Target_drawing_origin,-54,103,0),v50,fine,PencilHolder\WObj:=PAPER;
MoveL Offs(Target_drawing_origin,-54,178,0),v50,fine,PencilHolder\WObj:=PAPER;
MoveL Offs(Target_drawing_origin,-54,189,0),v50,fine,PencilHolder\WObj:=PAPER;
MoveL Offs(Target_drawing_origin,-54,216,0),v50,fine,PencilHolder\WObj:=PAPER;
MoveL Offs(Target_drawing_origin,-54,222,0),v50,fine,PencilHolder\WObj:=PAPER;
MoveL Offs(Target_drawing_origin,-54,248,0),v50,fine,PencilHolder\WObj:=PAPER;
MoveL Offs(Target_drawing_origin,-55,5,0),v50,fine,PencilHolder\WObj:=PAPER;
MoveL Offs(Target_drawing_origin,-55,37,0),v50,fine,PencilHolder\WObj:=PAPER;
MoveL Offs(Target_drawing_origin,-55,59,0),v50,fine,PencilHolder\WObj:=PAPER;
MoveL Offs(Target_drawing_origin,-55,91,0),v50,fine,PencilHolder\WObj:=PAPER;
MoveL Offs(Target_drawing_origin,-55,103,0),v50,fine,PencilHolder\WObj:=PAPER;
MoveL Offs(Target_drawing_origin,-55,178,0),v50,fine,PencilHolder\WObj:=PAPER;
MoveL Offs(Target_drawing_origin,-55,189,0),v50,fine,PencilHolder\WObj:=PAPER;
MoveL Offs(Target_drawing_origin,-55,216,0),v50,fine,PencilHolder\WObj:=PAPER;
MoveL Offs(Target_drawing_origin,-55,222,0),v50,fine,PencilHolder\WObj:=PAPER;
MoveL Offs(Target_drawing_origin,-55,248,0),v50,fine,PencilHolder\WObj:=PAPER;
MoveL Offs(Target_drawing_origin,-56,5,0),v50,fine,PencilHolder\WObj:=PAPER;
MoveL Offs(Target_drawing_origin,-56,37,0),v50,fine,PencilHolder\WObj:=PAPER;
MoveL Offs(Target_drawing_origin,-56,59,0),v50,fine,PencilHolder\WObj:=PAPER;
MoveL Offs(Target_drawing_origin,-56,91,0),v50,fine,PencilHolder\WObj:=PAPER;
MoveL Offs(Target_drawing_origin,-56,103,0),v50,fine,PencilHolder\WObj:=PAPER;
MoveL Offs(Target_drawing_origin,-56,178,0),v50,fine,PencilHolder\WObj:=PAPER;
MoveL Offs(Target_drawing_origin,-56,189,0),v50,fine,PencilHolder\WObj:=PAPER;
MoveL Offs(Target_drawing_origin,-56,216,0),v50,fine,PencilHolder\WObj:=PAPER;
MoveL Offs(Target_drawing_origin,-56,222,0),v50,fine,PencilHolder\WObj:=PAPER;
MoveL Offs(Target_drawing_origin,-56,248,0),v50,fine,PencilHolder\WObj:=PAPER;
MoveL Offs(Target_drawing_origin,-57,5,0),v50,fine,PencilHolder\WObj:=PAPER;
MoveL Offs(Target_drawing_origin,-57,37,0),v50,fine,PencilHolder\WObj:=PAPER;
MoveL Offs(Target_drawing_origin,-57,59,0),v50,fine,PencilHolder\WObj:=PAPER;
MoveL Offs(Target_drawing_origin,-57,91,0),v50,fine,PencilHolder\WObj:=PAPER;
MoveL Offs(Target_drawing_origin,-57,103,0),v50,fine,PencilHolder\WObj:=PAPER;
MoveL Offs(Target_drawing_origin,-57,178,0),v50,fine,PencilHolder\WObj:=PAPER;
MoveL Offs(Target_drawing_origin,-57,189,0),v50,fine,PencilHolder\WObj:=PAPER;
MoveL Offs(Target_drawing_origin,-57,216,0),v50,fine,PencilHolder\WObj:=PAPER;
MoveL Offs(Target_drawing_origin,-57,222,0),v50,fine,PencilHolder\WObj:=PAPER;
MoveL Offs(Target_drawing_origin,-57,248,0),v50,fine,PencilHolder\WObj:=PAPER;
MoveL Offs(Target_drawing_origin,-58,5,0),v50,fine,PencilHolder\WObj:=PAPER;
MoveL Offs(Target_drawing_origin,-58,37,0),v50,fine,PencilHolder\WObj:=PAPER;
MoveL Offs(Target_drawing_origin,-58,59,0),v50,fine,PencilHolder\WObj:=PAPER;
MoveL Offs(Target_drawing_origin,-58,91,0),v50,fine,PencilHolder\WObj:=PAPER;
MoveL Offs(Target_drawing_origin,-58,103,0),v50,fine,PencilHolder\WObj:=PAPER;
MoveL Offs(Target_drawing_origin,-58,178,0),v50,fine,PencilHolder\WObj:=PAPER;
MoveL Offs(Target_drawing_origin,-58,189,0),v50,fine,PencilHolder\WObj:=PAPER;
MoveL Offs(Target_drawing_origin,-58,216,0),v50,fine,PencilHolder\WObj:=PAPER;
MoveL Offs(Target_drawing_origin,-58,222,0),v50,fine,PencilHolder\WObj:=PAPER;
MoveL Offs(Target_drawing_origin,-58,248,0),v50,fine,PencilHolder\WObj:=PAPER;
MoveL Offs(Target_drawing_origin,-59,6,0),v50,fine,PencilHolder\WObj:=PAPER;
MoveL Offs(Target_drawing_origin,-59,37,0),v50,fine,PencilHolder\WObj:=PAPER;
MoveL Offs(Target_drawing_origin,-59,54,0),v50,fine,PencilHolder\WObj:=PAPER;
MoveL Offs(Target_drawing_origin,-59,91,0),v50,fine,PencilHolder\WObj:=PAPER;
MoveL Offs(Target_drawing_origin,-59,103,0),v50,fine,PencilHolder\WObj:=PAPER;
MoveL Offs(Target_drawing_origin,-59,183,0),v50,fine,PencilHolder\WObj:=PAPER;
MoveL Offs(Target_drawing_origin,-59,189,0),v50,fine,PencilHolder\WObj:=PAPER;
MoveL Offs(Target_drawing_origin,-59,216,0),v50,fine,PencilHolder\WObj:=PAPER;
MoveL Offs(Target_drawing_origin,-59,222,0),v50,fine,PencilHolder\WObj:=PAPER;
MoveL Offs(Target_drawing_origin,-59,248,0),v50,fine,PencilHolder\WObj:=PAPER;
MoveL Offs(Target_drawing_origin,-60,54,0),v50,fine,PencilHolder\WObj:=PAPER;
MoveL Offs(Target_drawing_origin,-60,91,0),v50,fine,PencilHolder\WObj:=PAPER;
MoveL Offs(Target_drawing_origin,-60,103,0),v50,fine,PencilHolder\WObj:=PAPER;
MoveL Offs(Target_drawing_origin,-60,130,0),v50,fine,PencilHolder\WObj:=PAPER;
MoveL Offs(Target_drawing_origin,-60,146,0),v50,fine,PencilHolder\WObj:=PAPER;
MoveL Offs(Target_drawing_origin,-60,183,0),v50,fine,PencilHolder\WObj:=PAPER;
MoveL Offs(Target_drawing_origin,-60,189,0),v50,fine,PencilHolder\WObj:=PAPER;
MoveL Offs(Target_drawing_origin,-60,216,0),v50,fine,PencilHolder\WObj:=PAPER;
MoveL Offs(Target_drawing_origin,-60,222,0),v50,fine,PencilHolder\WObj:=PAPER;
MoveL Offs(Target_drawing_origin,-60,248,0),v50,fine,PencilHolder\WObj:=PAPER;
MoveL Offs(Target_drawing_origin,-61,54,0),v50,fine,PencilHolder\WObj:=PAPER;
MoveL Offs(Target_drawing_origin,-61,91,0),v50,fine,PencilHolder\WObj:=PAPER;
MoveL Offs(Target_drawing_origin,-61,103,0),v50,fine,PencilHolder\WObj:=PAPER;
MoveL Offs(Target_drawing_origin,-61,130,0),v50,fine,PencilHolder\WObj:=PAPER;
MoveL Offs(Target_drawing_origin,-61,146,0),v50,fine,PencilHolder\WObj:=PAPER;
MoveL Offs(Target_drawing_origin,-61,183,0),v50,fine,PencilHolder\WObj:=PAPER;
MoveL Offs(Target_drawing_origin,-61,189,0),v50,fine,PencilHolder\WObj:=PAPER;
MoveL Offs(Target_drawing_origin,-61,216,0),v50,fine,PencilHolder\WObj:=PAPER;
MoveL Offs(Target_drawing_origin,-61,222,0),v50,fine,PencilHolder\WObj:=PAPER;
MoveL Offs(Target_drawing_origin,-61,248,0),v50,fine,PencilHolder\WObj:=PAPER;
MoveL Offs(Target_drawing_origin,-62,54,0),v50,fine,PencilHolder\WObj:=PAPER;
MoveL Offs(Target_drawing_origin,-62,91,0),v50,fine,PencilHolder\WObj:=PAPER;
MoveL Offs(Target_drawing_origin,-62,103,0),v50,fine,PencilHolder\WObj:=PAPER;
MoveL Offs(Target_drawing_origin,-62,130,0),v50,fine,PencilHolder\WObj:=PAPER;
MoveL Offs(Target_drawing_origin,-62,146,0),v50,fine,PencilHolder\WObj:=PAPER;
MoveL Offs(Target_drawing_origin,-62,183,0),v50,fine,PencilHolder\WObj:=PAPER;
MoveL Offs(Target_drawing_origin,-62,189,0),v50,fine,PencilHolder\WObj:=PAPER;
MoveL Offs(Target_drawing_origin,-62,216,0),v50,fine,PencilHolder\WObj:=PAPER;
MoveL Offs(Target_drawing_origin,-62,222,0),v50,fine,PencilHolder\WObj:=PAPER;
MoveL Offs(Target_drawing_origin,-62,248,0),v50,fine,PencilHolder\WObj:=PAPER;
MoveL Offs(Target_drawing_origin,-63,54,0),v50,fine,PencilHolder\WObj:=PAPER;
MoveL Offs(Target_drawing_origin,-63,91,0),v50,fine,PencilHolder\WObj:=PAPER;
MoveL Offs(Target_drawing_origin,-63,103,0),v50,fine,PencilHolder\WObj:=PAPER;
MoveL Offs(Target_drawing_origin,-63,130,0),v50,fine,PencilHolder\WObj:=PAPER;
MoveL Offs(Target_drawing_origin,-63,146,0),v50,fine,PencilHolder\WObj:=PAPER;
MoveL Offs(Target_drawing_origin,-63,183,0),v50,fine,PencilHolder\WObj:=PAPER;
MoveL Offs(Target_drawing_origin,-63,189,0),v50,fine,PencilHolder\WObj:=PAPER;
MoveL Offs(Target_drawing_origin,-63,216,0),v50,fine,PencilHolder\WObj:=PAPER;
MoveL Offs(Target_drawing_origin,-63,222,0),v50,fine,PencilHolder\WObj:=PAPER;
MoveL Offs(Target_drawing_origin,-63,248,0),v50,fine,PencilHolder\WObj:=PAPER;
MoveL Offs(Target_drawing_origin,-64,54,0),v50,fine,PencilHolder\WObj:=PAPER;
MoveL Offs(Target_drawing_origin,-64,91,0),v50,fine,PencilHolder\WObj:=PAPER;
MoveL Offs(Target_drawing_origin,-64,103,0),v50,fine,PencilHolder\WObj:=PAPER;
MoveL Offs(Target_drawing_origin,-64,130,0),v50,fine,PencilHolder\WObj:=PAPER;
MoveL Offs(Target_drawing_origin,-64,146,0),v50,fine,PencilHolder\WObj:=PAPER;
MoveL Offs(Target_drawing_origin,-64,183,0),v50,fine,PencilHolder\WObj:=PAPER;
MoveL Offs(Target_drawing_origin,-64,189,0),v50,fine,PencilHolder\WObj:=PAPER;
MoveL Offs(Target_drawing_origin,-64,216,0),v50,fine,PencilHolder\WObj:=PAPER;
MoveL Offs(Target_drawing_origin,-64,222,0),v50,fine,PencilHolder\WObj:=PAPER;
MoveL Offs(Target_drawing_origin,-64,248,0),v50,fine,PencilHolder\WObj:=PAPER;
MoveL Offs(Target_drawing_origin,-65,54,0),v50,fine,PencilHolder\WObj:=PAPER;
MoveL Offs(Target_drawing_origin,-65,86,0),v50,fine,PencilHolder\WObj:=PAPER;
MoveL Offs(Target_drawing_origin,-65,97,0),v50,fine,PencilHolder\WObj:=PAPER;
MoveL Offs(Target_drawing_origin,-65,130,0),v50,fine,PencilHolder\WObj:=PAPER;
MoveL Offs(Target_drawing_origin,-65,152,0),v50,fine,PencilHolder\WObj:=PAPER;
MoveL Offs(Target_drawing_origin,-65,183,0),v50,fine,PencilHolder\WObj:=PAPER;
MoveL Offs(Target_drawing_origin,-65,189,0),v50,fine,PencilHolder\WObj:=PAPER;
MoveL Offs(Target_drawing_origin,-65,210,0),v50,fine,PencilHolder\WObj:=PAPER;
MoveL Offs(Target_drawing_origin,-65,222,0),v50,fine,PencilHolder\WObj:=PAPER;
MoveL Offs(Target_drawing_origin,-65,248,0),v50,fine,PencilHolder\WObj:=PAPER;
MoveL Offs(Target_drawing_origin,-66,54,0),v50,fine,PencilHolder\WObj:=PAPER;
MoveL Offs(Target_drawing_origin,-66,86,0),v50,fine,PencilHolder\WObj:=PAPER;
MoveL Offs(Target_drawing_origin,-66,97,0),v50,fine,PencilHolder\WObj:=PAPER;
MoveL Offs(Target_drawing_origin,-66,130,0),v50,fine,PencilHolder\WObj:=PAPER;
MoveL Offs(Target_drawing_origin,-66,152,0),v50,fine,PencilHolder\WObj:=PAPER;
MoveL Offs(Target_drawing_origin,-66,183,0),v50,fine,PencilHolder\WObj:=PAPER;
MoveL Offs(Target_drawing_origin,-66,189,0),v50,fine,PencilHolder\WObj:=PAPER;
MoveL Offs(Target_drawing_origin,-66,210,0),v50,fine,PencilHolder\WObj:=PAPER;
MoveL Offs(Target_drawing_origin,-66,222,0),v50,fine,PencilHolder\WObj:=PAPER;
MoveL Offs(Target_drawing_origin,-66,248,0),v50,fine,PencilHolder\WObj:=PAPER;
MoveL Offs(Target_drawing_origin,-67,54,0),v50,fine,PencilHolder\WObj:=PAPER;
MoveL Offs(Target_drawing_origin,-67,86,0),v50,fine,PencilHolder\WObj:=PAPER;
MoveL Offs(Target_drawing_origin,-67,97,0),v50,fine,PencilHolder\WObj:=PAPER;
MoveL Offs(Target_drawing_origin,-67,130,0),v50,fine,PencilHolder\WObj:=PAPER;
MoveL Offs(Target_drawing_origin,-67,152,0),v50,fine,PencilHolder\WObj:=PAPER;
MoveL Offs(Target_drawing_origin,-67,183,0),v50,fine,PencilHolder\WObj:=PAPER;
MoveL Offs(Target_drawing_origin,-67,189,0),v50,fine,PencilHolder\WObj:=PAPER;
MoveL Offs(Target_drawing_origin,-67,210,0),v50,fine,PencilHolder\WObj:=PAPER;
MoveL Offs(Target_drawing_origin,-67,222,0),v50,fine,PencilHolder\WObj:=PAPER;
MoveL Offs(Target_drawing_origin,-67,248,0),v50,fine,PencilHolder\WObj:=PAPER;
MoveL Offs(Target_drawing_origin,-68,54,0),v50,fine,PencilHolder\WObj:=PAPER;
MoveL Offs(Target_drawing_origin,-68,86,0),v50,fine,PencilHolder\WObj:=PAPER;
MoveL Offs(Target_drawing_origin,-68,97,0),v50,fine,PencilHolder\WObj:=PAPER;
MoveL Offs(Target_drawing_origin,-68,130,0),v50,fine,PencilHolder\WObj:=PAPER;
MoveL Offs(Target_drawing_origin,-68,152,0),v50,fine,PencilHolder\WObj:=PAPER;
MoveL Offs(Target_drawing_origin,-68,183,0),v50,fine,PencilHolder\WObj:=PAPER;
MoveL Offs(Target_drawing_origin,-68,189,0),v50,fine,PencilHolder\WObj:=PAPER;
MoveL Offs(Target_drawing_origin,-68,210,0),v50,fine,PencilHolder\WObj:=PAPER;
MoveL Offs(Target_drawing_origin,-68,222,0),v50,fine,PencilHolder\WObj:=PAPER;
MoveL Offs(Target_drawing_origin,-68,248,0),v50,fine,PencilHolder\WObj:=PAPER;
MoveL Offs(Target_drawing_origin,-69,54,0),v50,fine,PencilHolder\WObj:=PAPER;
MoveL Offs(Target_drawing_origin,-69,86,0),v50,fine,PencilHolder\WObj:=PAPER;
MoveL Offs(Target_drawing_origin,-69,97,0),v50,fine,PencilHolder\WObj:=PAPER;
MoveL Offs(Target_drawing_origin,-69,130,0),v50,fine,PencilHolder\WObj:=PAPER;
MoveL Offs(Target_drawing_origin,-69,152,0),v50,fine,PencilHolder\WObj:=PAPER;
MoveL Offs(Target_drawing_origin,-69,183,0),v50,fine,PencilHolder\WObj:=PAPER;
MoveL Offs(Target_drawing_origin,-69,189,0),v50,fine,PencilHolder\WObj:=PAPER;
MoveL Offs(Target_drawing_origin,-69,210,0),v50,fine,PencilHolder\WObj:=PAPER;
MoveL Offs(Target_drawing_origin,-69,222,0),v50,fine,PencilHolder\WObj:=PAPER;
MoveL Offs(Target_drawing_origin,-69,248,0),v50,fine,PencilHolder\WObj:=PAPER;
MoveL Offs(Target_drawing_origin,-70,49,0),v50,fine,PencilHolder\WObj:=PAPER;
MoveL Offs(Target_drawing_origin,-70,81,0),v50,fine,PencilHolder\WObj:=PAPER;
MoveL Offs(Target_drawing_origin,-70,97,0),v50,fine,PencilHolder\WObj:=PAPER;
MoveL Offs(Target_drawing_origin,-70,124,0),v50,fine,PencilHolder\WObj:=PAPER;
MoveL Offs(Target_drawing_origin,-70,157,0),v50,fine,PencilHolder\WObj:=PAPER;
MoveL Offs(Target_drawing_origin,-70,183,0),v50,fine,PencilHolder\WObj:=PAPER;
MoveL Offs(Target_drawing_origin,-70,189,0),v50,fine,PencilHolder\WObj:=PAPER;
MoveL Offs(Target_drawing_origin,-70,216,0),v50,fine,PencilHolder\WObj:=PAPER;
MoveL Offs(Target_drawing_origin,-70,227,0),v50,fine,PencilHolder\WObj:=PAPER;
MoveL Offs(Target_drawing_origin,-70,248,0),v50,fine,PencilHolder\WObj:=PAPER;
MoveL Offs(Target_drawing_origin,-71,49,0),v50,fine,PencilHolder\WObj:=PAPER;
MoveL Offs(Target_drawing_origin,-71,80,0),v50,fine,PencilHolder\WObj:=PAPER;
MoveL Offs(Target_drawing_origin,-71,97,0),v50,fine,PencilHolder\WObj:=PAPER;
MoveL Offs(Target_drawing_origin,-71,124,0),v50,fine,PencilHolder\WObj:=PAPER;
MoveL Offs(Target_drawing_origin,-71,157,0),v50,fine,PencilHolder\WObj:=PAPER;
MoveL Offs(Target_drawing_origin,-71,183,0),v50,fine,PencilHolder\WObj:=PAPER;
MoveL Offs(Target_drawing_origin,-71,189,0),v50,fine,PencilHolder\WObj:=PAPER;
MoveL Offs(Target_drawing_origin,-71,216,0),v50,fine,PencilHolder\WObj:=PAPER;
MoveL Offs(Target_drawing_origin,-71,227,0),v50,fine,PencilHolder\WObj:=PAPER;
MoveL Offs(Target_drawing_origin,-71,248,0),v50,fine,PencilHolder\WObj:=PAPER;
MoveL Offs(Target_drawing_origin,-72,49,0),v50,fine,PencilHolder\WObj:=PAPER;
MoveL Offs(Target_drawing_origin,-72,80,0),v50,fine,PencilHolder\WObj:=PAPER;
MoveL Offs(Target_drawing_origin,-72,97,0),v50,fine,PencilHolder\WObj:=PAPER;
MoveL Offs(Target_drawing_origin,-72,124,0),v50,fine,PencilHolder\WObj:=PAPER;
MoveL Offs(Target_drawing_origin,-72,157,0),v50,fine,PencilHolder\WObj:=PAPER;
MoveL Offs(Target_drawing_origin,-72,183,0),v50,fine,PencilHolder\WObj:=PAPER;
MoveL Offs(Target_drawing_origin,-72,189,0),v50,fine,PencilHolder\WObj:=PAPER;
MoveL Offs(Target_drawing_origin,-72,216,0),v50,fine,PencilHolder\WObj:=PAPER;
MoveL Offs(Target_drawing_origin,-72,227,0),v50,fine,PencilHolder\WObj:=PAPER;
MoveL Offs(Target_drawing_origin,-72,248,0),v50,fine,PencilHolder\WObj:=PAPER;
MoveL Offs(Target_drawing_origin,-73,49,0),v50,fine,PencilHolder\WObj:=PAPER;
MoveL Offs(Target_drawing_origin,-73,80,0),v50,fine,PencilHolder\WObj:=PAPER;
MoveL Offs(Target_drawing_origin,-73,97,0),v50,fine,PencilHolder\WObj:=PAPER;
MoveL Offs(Target_drawing_origin,-73,124,0),v50,fine,PencilHolder\WObj:=PAPER;
MoveL Offs(Target_drawing_origin,-73,157,0),v50,fine,PencilHolder\WObj:=PAPER;
MoveL Offs(Target_drawing_origin,-73,183,0),v50,fine,PencilHolder\WObj:=PAPER;
MoveL Offs(Target_drawing_origin,-73,189,0),v50,fine,PencilHolder\WObj:=PAPER;
MoveL Offs(Target_drawing_origin,-73,216,0),v50,fine,PencilHolder\WObj:=PAPER;
MoveL Offs(Target_drawing_origin,-73,227,0),v50,fine,PencilHolder\WObj:=PAPER;
MoveL Offs(Target_drawing_origin,-73,248,0),v50,fine,PencilHolder\WObj:=PAPER;
MoveL Offs(Target_drawing_origin,-74,49,0),v50,fine,PencilHolder\WObj:=PAPER;
MoveL Offs(Target_drawing_origin,-74,80,0),v50,fine,PencilHolder\WObj:=PAPER;
MoveL Offs(Target_drawing_origin,-74,97,0),v50,fine,PencilHolder\WObj:=PAPER;
MoveL Offs(Target_drawing_origin,-74,124,0),v50,fine,PencilHolder\WObj:=PAPER;
MoveL Offs(Target_drawing_origin,-74,157,0),v50,fine,PencilHolder\WObj:=PAPER;
MoveL Offs(Target_drawing_origin,-74,183,0),v50,fine,PencilHolder\WObj:=PAPER;
MoveL Offs(Target_drawing_origin,-74,189,0),v50,fine,PencilHolder\WObj:=PAPER;
MoveL Offs(Target_drawing_origin,-74,216,0),v50,fine,PencilHolder\WObj:=PAPER;
MoveL Offs(Target_drawing_origin,-74,227,0),v50,fine,PencilHolder\WObj:=PAPER;
MoveL Offs(Target_drawing_origin,-74,248,0),v50,fine,PencilHolder\WObj:=PAPER;
MoveL Offs(Target_drawing_origin,-75,48,0),v50,fine,PencilHolder\WObj:=PAPER;
MoveL Offs(Target_drawing_origin,-75,80,0),v50,fine,PencilHolder\WObj:=PAPER;
MoveL Offs(Target_drawing_origin,-75,97,0),v50,fine,PencilHolder\WObj:=PAPER;
MoveL Offs(Target_drawing_origin,-75,124,0),v50,fine,PencilHolder\WObj:=PAPER;
MoveL Offs(Target_drawing_origin,-75,157,0),v50,fine,PencilHolder\WObj:=PAPER;
MoveL Offs(Target_drawing_origin,-75,183,0),v50,fine,PencilHolder\WObj:=PAPER;
MoveL Offs(Target_drawing_origin,-75,189,0),v50,fine,PencilHolder\WObj:=PAPER;
MoveL Offs(Target_drawing_origin,-75,216,0),v50,fine,PencilHolder\WObj:=PAPER;
MoveL Offs(Target_drawing_origin,-75,227,0),v50,fine,PencilHolder\WObj:=PAPER;
MoveL Offs(Target_drawing_origin,-75,248,0),v50,fine,PencilHolder\WObj:=PAPER;
MoveL Offs(Target_drawing_origin,-76,43,0),v50,fine,PencilHolder\WObj:=PAPER;
MoveL Offs(Target_drawing_origin,-76,75,0),v50,fine,PencilHolder\WObj:=PAPER;
MoveL Offs(Target_drawing_origin,-76,97,0),v50,fine,PencilHolder\WObj:=PAPER;
MoveL Offs(Target_drawing_origin,-76,124,0),v50,fine,PencilHolder\WObj:=PAPER;
MoveL Offs(Target_drawing_origin,-76,157,0),v50,fine,PencilHolder\WObj:=PAPER;
MoveL Offs(Target_drawing_origin,-76,183,0),v50,fine,PencilHolder\WObj:=PAPER;
MoveL Offs(Target_drawing_origin,-76,189,0),v50,fine,PencilHolder\WObj:=PAPER;
MoveL Offs(Target_drawing_origin,-76,216,0),v50,fine,PencilHolder\WObj:=PAPER;
MoveL Offs(Target_drawing_origin,-76,227,0),v50,fine,PencilHolder\WObj:=PAPER;
MoveL Offs(Target_drawing_origin,-76,248,0),v50,fine,PencilHolder\WObj:=PAPER;
MoveL Offs(Target_drawing_origin,-77,43,0),v50,fine,PencilHolder\WObj:=PAPER;
MoveL Offs(Target_drawing_origin,-77,75,0),v50,fine,PencilHolder\WObj:=PAPER;
MoveL Offs(Target_drawing_origin,-77,97,0),v50,fine,PencilHolder\WObj:=PAPER;
MoveL Offs(Target_drawing_origin,-77,124,0),v50,fine,PencilHolder\WObj:=PAPER;
MoveL Offs(Target_drawing_origin,-77,157,0),v50,fine,PencilHolder\WObj:=PAPER;
MoveL Offs(Target_drawing_origin,-77,183,0),v50,fine,PencilHolder\WObj:=PAPER;
MoveL Offs(Target_drawing_origin,-77,189,0),v50,fine,PencilHolder\WObj:=PAPER;
MoveL Offs(Target_drawing_origin,-77,216,0),v50,fine,PencilHolder\WObj:=PAPER;
MoveL Offs(Target_drawing_origin,-77,227,0),v50,fine,PencilHolder\WObj:=PAPER;
MoveL Offs(Target_drawing_origin,-77,248,0),v50,fine,PencilHolder\WObj:=PAPER;
MoveL Offs(Target_drawing_origin,-78,43,0),v50,fine,PencilHolder\WObj:=PAPER;
MoveL Offs(Target_drawing_origin,-78,75,0),v50,fine,PencilHolder\WObj:=PAPER;
MoveL Offs(Target_drawing_origin,-78,97,0),v50,fine,PencilHolder\WObj:=PAPER;
MoveL Offs(Target_drawing_origin,-78,124,0),v50,fine,PencilHolder\WObj:=PAPER;
MoveL Offs(Target_drawing_origin,-78,157,0),v50,fine,PencilHolder\WObj:=PAPER;
MoveL Offs(Target_drawing_origin,-78,183,0),v50,fine,PencilHolder\WObj:=PAPER;
MoveL Offs(Target_drawing_origin,-78,189,0),v50,fine,PencilHolder\WObj:=PAPER;
MoveL Offs(Target_drawing_origin,-78,216,0),v50,fine,PencilHolder\WObj:=PAPER;
MoveL Offs(Target_drawing_origin,-78,227,0),v50,fine,PencilHolder\WObj:=PAPER;
MoveL Offs(Target_drawing_origin,-78,248,0),v50,fine,PencilHolder\WObj:=PAPER;
MoveL Offs(Target_drawing_origin,-79,43,0),v50,fine,PencilHolder\WObj:=PAPER;
MoveL Offs(Target_drawing_origin,-79,75,0),v50,fine,PencilHolder\WObj:=PAPER;
MoveL Offs(Target_drawing_origin,-79,97,0),v50,fine,PencilHolder\WObj:=PAPER;
MoveL Offs(Target_drawing_origin,-79,124,0),v50,fine,PencilHolder\WObj:=PAPER;
MoveL Offs(Target_drawing_origin,-79,157,0),v50,fine,PencilHolder\WObj:=PAPER;
MoveL Offs(Target_drawing_origin,-79,183,0),v50,fine,PencilHolder\WObj:=PAPER;
MoveL Offs(Target_drawing_origin,-79,189,0),v50,fine,PencilHolder\WObj:=PAPER;
MoveL Offs(Target_drawing_origin,-79,216,0),v50,fine,PencilHolder\WObj:=PAPER;
MoveL Offs(Target_drawing_origin,-79,227,0),v50,fine,PencilHolder\WObj:=PAPER;
MoveL Offs(Target_drawing_origin,-79,248,0),v50,fine,PencilHolder\WObj:=PAPER;
MoveL Offs(Target_drawing_origin,-80,43,0),v50,fine,PencilHolder\WObj:=PAPER;
MoveL Offs(Target_drawing_origin,-80,75,0),v50,fine,PencilHolder\WObj:=PAPER;
MoveL Offs(Target_drawing_origin,-80,97,0),v50,fine,PencilHolder\WObj:=PAPER;
MoveL Offs(Target_drawing_origin,-80,124,0),v50,fine,PencilHolder\WObj:=PAPER;
MoveL Offs(Target_drawing_origin,-80,157,0),v50,fine,PencilHolder\WObj:=PAPER;
MoveL Offs(Target_drawing_origin,-80,183,0),v50,fine,PencilHolder\WObj:=PAPER;
MoveL Offs(Target_drawing_origin,-80,189,0),v50,fine,PencilHolder\WObj:=PAPER;
MoveL Offs(Target_drawing_origin,-80,216,0),v50,fine,PencilHolder\WObj:=PAPER;
MoveL Offs(Target_drawing_origin,-80,227,0),v50,fine,PencilHolder\WObj:=PAPER;
MoveL Offs(Target_drawing_origin,-80,248,0),v50,fine,PencilHolder\WObj:=PAPER;
MoveL Offs(Target_drawing_origin,-81,43,0),v50,fine,PencilHolder\WObj:=PAPER;
MoveL Offs(Target_drawing_origin,-81,75,0),v50,fine,PencilHolder\WObj:=PAPER;
MoveL Offs(Target_drawing_origin,-81,92,0),v50,fine,PencilHolder\WObj:=PAPER;
MoveL Offs(Target_drawing_origin,-81,124,0),v50,fine,PencilHolder\WObj:=PAPER;
MoveL Offs(Target_drawing_origin,-81,157,0),v50,fine,PencilHolder\WObj:=PAPER;
MoveL Offs(Target_drawing_origin,-81,183,0),v50,fine,PencilHolder\WObj:=PAPER;
MoveL Offs(Target_drawing_origin,-81,189,0),v50,fine,PencilHolder\WObj:=PAPER;
MoveL Offs(Target_drawing_origin,-81,216,0),v50,fine,PencilHolder\WObj:=PAPER;
MoveL Offs(Target_drawing_origin,-81,227,0),v50,fine,PencilHolder\WObj:=PAPER;
MoveL Offs(Target_drawing_origin,-81,248,0),v50,fine,PencilHolder\WObj:=PAPER;
MoveL Offs(Target_drawing_origin,-82,43,0),v50,fine,PencilHolder\WObj:=PAPER;
MoveL Offs(Target_drawing_origin,-82,75,0),v50,fine,PencilHolder\WObj:=PAPER;
MoveL Offs(Target_drawing_origin,-82,92,0),v50,fine,PencilHolder\WObj:=PAPER;
MoveL Offs(Target_drawing_origin,-82,124,0),v50,fine,PencilHolder\WObj:=PAPER;
MoveL Offs(Target_drawing_origin,-82,157,0),v50,fine,PencilHolder\WObj:=PAPER;
MoveL Offs(Target_drawing_origin,-82,183,0),v50,fine,PencilHolder\WObj:=PAPER;
MoveL Offs(Target_drawing_origin,-82,189,0),v50,fine,PencilHolder\WObj:=PAPER;
MoveL Offs(Target_drawing_origin,-82,216,0),v50,fine,PencilHolder\WObj:=PAPER;
MoveL Offs(Target_drawing_origin,-82,227,0),v50,fine,PencilHolder\WObj:=PAPER;
MoveL Offs(Target_drawing_origin,-82,248,0),v50,fine,PencilHolder\WObj:=PAPER;
MoveL Offs(Target_drawing_origin,-83,43,0),v50,fine,PencilHolder\WObj:=PAPER;
MoveL Offs(Target_drawing_origin,-83,75,0),v50,fine,PencilHolder\WObj:=PAPER;
MoveL Offs(Target_drawing_origin,-83,92,0),v50,fine,PencilHolder\WObj:=PAPER;
MoveL Offs(Target_drawing_origin,-83,124,0),v50,fine,PencilHolder\WObj:=PAPER;
MoveL Offs(Target_drawing_origin,-83,157,0),v50,fine,PencilHolder\WObj:=PAPER;
MoveL Offs(Target_drawing_origin,-83,183,0),v50,fine,PencilHolder\WObj:=PAPER;
MoveL Offs(Target_drawing_origin,-83,189,0),v50,fine,PencilHolder\WObj:=PAPER;
MoveL Offs(Target_drawing_origin,-83,216,0),v50,fine,PencilHolder\WObj:=PAPER;
MoveL Offs(Target_drawing_origin,-83,227,0),v50,fine,PencilHolder\WObj:=PAPER;
MoveL Offs(Target_drawing_origin,-83,248,0),v50,fine,PencilHolder\WObj:=PAPER;
MoveL Offs(Target_drawing_origin,-84,43,0),v50,fine,PencilHolder\WObj:=PAPER;
MoveL Offs(Target_drawing_origin,-84,75,0),v50,fine,PencilHolder\WObj:=PAPER;
MoveL Offs(Target_drawing_origin,-84,92,0),v50,fine,PencilHolder\WObj:=PAPER;
MoveL Offs(Target_drawing_origin,-84,124,0),v50,fine,PencilHolder\WObj:=PAPER;
MoveL Offs(Target_drawing_origin,-84,157,0),v50,fine,PencilHolder\WObj:=PAPER;
MoveL Offs(Target_drawing_origin,-84,183,0),v50,fine,PencilHolder\WObj:=PAPER;
MoveL Offs(Target_drawing_origin,-84,189,0),v50,fine,PencilHolder\WObj:=PAPER;
MoveL Offs(Target_drawing_origin,-84,216,0),v50,fine,PencilHolder\WObj:=PAPER;
MoveL Offs(Target_drawing_origin,-84,227,0),v50,fine,PencilHolder\WObj:=PAPER;
MoveL Offs(Target_drawing_origin,-84,248,0),v50,fine,PencilHolder\WObj:=PAPER;
MoveL Offs(Target_drawing_origin,-85,43,0),v50,fine,PencilHolder\WObj:=PAPER;
MoveL Offs(Target_drawing_origin,-85,75,0),v50,fine,PencilHolder\WObj:=PAPER;
MoveL Offs(Target_drawing_origin,-85,92,0),v50,fine,PencilHolder\WObj:=PAPER;
MoveL Offs(Target_drawing_origin,-85,124,0),v50,fine,PencilHolder\WObj:=PAPER;
MoveL Offs(Target_drawing_origin,-85,157,0),v50,fine,PencilHolder\WObj:=PAPER;
MoveL Offs(Target_drawing_origin,-85,183,0),v50,fine,PencilHolder\WObj:=PAPER;
MoveL Offs(Target_drawing_origin,-85,189,0),v50,fine,PencilHolder\WObj:=PAPER;
MoveL Offs(Target_drawing_origin,-85,216,0),v50,fine,PencilHolder\WObj:=PAPER;
MoveL Offs(Target_drawing_origin,-85,227,0),v50,fine,PencilHolder\WObj:=PAPER;
MoveL Offs(Target_drawing_origin,-85,248,0),v50,fine,PencilHolder\WObj:=PAPER;
MoveL Offs(Target_drawing_origin,-86,43,0),v50,fine,PencilHolder\WObj:=PAPER;
MoveL Offs(Target_drawing_origin,-86,75,0),v50,fine,PencilHolder\WObj:=PAPER;
MoveL Offs(Target_drawing_origin,-86,87,0),v50,fine,PencilHolder\WObj:=PAPER;
MoveL Offs(Target_drawing_origin,-86,123,0),v50,fine,PencilHolder\WObj:=PAPER;
MoveL Offs(Target_drawing_origin,-86,157,0),v50,fine,PencilHolder\WObj:=PAPER;
MoveL Offs(Target_drawing_origin,-86,183,0),v50,fine,PencilHolder\WObj:=PAPER;
MoveL Offs(Target_drawing_origin,-86,190,0),v50,fine,PencilHolder\WObj:=PAPER;
MoveL Offs(Target_drawing_origin,-86,216,0),v50,fine,PencilHolder\WObj:=PAPER;
MoveL Offs(Target_drawing_origin,-86,227,0),v50,fine,PencilHolder\WObj:=PAPER;
MoveL Offs(Target_drawing_origin,-86,248,0),v50,fine,PencilHolder\WObj:=PAPER;
MoveL Offs(Target_drawing_origin,-87,43,0),v50,fine,PencilHolder\WObj:=PAPER;
MoveL Offs(Target_drawing_origin,-87,75,0),v50,fine,PencilHolder\WObj:=PAPER;
MoveL Offs(Target_drawing_origin,-87,87,0),v50,fine,PencilHolder\WObj:=PAPER;
MoveL Offs(Target_drawing_origin,-87,118,0),v50,fine,PencilHolder\WObj:=PAPER;
MoveL Offs(Target_drawing_origin,-87,157,0),v50,fine,PencilHolder\WObj:=PAPER;
MoveL Offs(Target_drawing_origin,-87,183,0),v50,fine,PencilHolder\WObj:=PAPER;
MoveL Offs(Target_drawing_origin,-87,195,0),v50,fine,PencilHolder\WObj:=PAPER;
MoveL Offs(Target_drawing_origin,-87,216,0),v50,fine,PencilHolder\WObj:=PAPER;
MoveL Offs(Target_drawing_origin,-87,227,0),v50,fine,PencilHolder\WObj:=PAPER;
MoveL Offs(Target_drawing_origin,-87,248,0),v50,fine,PencilHolder\WObj:=PAPER;
MoveL Offs(Target_drawing_origin,-88,43,0),v50,fine,PencilHolder\WObj:=PAPER;
MoveL Offs(Target_drawing_origin,-88,75,0),v50,fine,PencilHolder\WObj:=PAPER;
MoveL Offs(Target_drawing_origin,-88,87,0),v50,fine,PencilHolder\WObj:=PAPER;
MoveL Offs(Target_drawing_origin,-88,118,0),v50,fine,PencilHolder\WObj:=PAPER;
MoveL Offs(Target_drawing_origin,-88,157,0),v50,fine,PencilHolder\WObj:=PAPER;
MoveL Offs(Target_drawing_origin,-88,183,0),v50,fine,PencilHolder\WObj:=PAPER;
MoveL Offs(Target_drawing_origin,-88,195,0),v50,fine,PencilHolder\WObj:=PAPER;
MoveL Offs(Target_drawing_origin,-88,216,0),v50,fine,PencilHolder\WObj:=PAPER;
MoveL Offs(Target_drawing_origin,-88,227,0),v50,fine,PencilHolder\WObj:=PAPER;
MoveL Offs(Target_drawing_origin,-88,248,0),v50,fine,PencilHolder\WObj:=PAPER;
MoveL Offs(Target_drawing_origin,-89,43,0),v50,fine,PencilHolder\WObj:=PAPER;
MoveL Offs(Target_drawing_origin,-89,75,0),v50,fine,PencilHolder\WObj:=PAPER;
MoveL Offs(Target_drawing_origin,-89,87,0),v50,fine,PencilHolder\WObj:=PAPER;
MoveL Offs(Target_drawing_origin,-89,118,0),v50,fine,PencilHolder\WObj:=PAPER;
MoveL Offs(Target_drawing_origin,-89,157,0),v50,fine,PencilHolder\WObj:=PAPER;
MoveL Offs(Target_drawing_origin,-89,183,0),v50,fine,PencilHolder\WObj:=PAPER;
MoveL Offs(Target_drawing_origin,-89,195,0),v50,fine,PencilHolder\WObj:=PAPER;
MoveL Offs(Target_drawing_origin,-89,216,0),v50,fine,PencilHolder\WObj:=PAPER;
MoveL Offs(Target_drawing_origin,-89,227,0),v50,fine,PencilHolder\WObj:=PAPER;
MoveL Offs(Target_drawing_origin,-89,248,0),v50,fine,PencilHolder\WObj:=PAPER;
MoveL Offs(Target_drawing_origin,-90,43,0),v50,fine,PencilHolder\WObj:=PAPER;
MoveL Offs(Target_drawing_origin,-90,75,0),v50,fine,PencilHolder\WObj:=PAPER;
MoveL Offs(Target_drawing_origin,-90,87,0),v50,fine,PencilHolder\WObj:=PAPER;
MoveL Offs(Target_drawing_origin,-90,118,0),v50,fine,PencilHolder\WObj:=PAPER;
MoveL Offs(Target_drawing_origin,-90,157,0),v50,fine,PencilHolder\WObj:=PAPER;
MoveL Offs(Target_drawing_origin,-90,183,0),v50,fine,PencilHolder\WObj:=PAPER;
MoveL Offs(Target_drawing_origin,-90,195,0),v50,fine,PencilHolder\WObj:=PAPER;
MoveL Offs(Target_drawing_origin,-90,216,0),v50,fine,PencilHolder\WObj:=PAPER;
MoveL Offs(Target_drawing_origin,-90,227,0),v50,fine,PencilHolder\WObj:=PAPER;
MoveL Offs(Target_drawing_origin,-90,248,0),v50,fine,PencilHolder\WObj:=PAPER;
MoveL Offs(Target_drawing_origin,-91,43,0),v50,fine,PencilHolder\WObj:=PAPER;
MoveL Offs(Target_drawing_origin,-91,75,0),v50,fine,PencilHolder\WObj:=PAPER;
MoveL Offs(Target_drawing_origin,-91,87,0),v50,fine,PencilHolder\WObj:=PAPER;
MoveL Offs(Target_drawing_origin,-91,118,0),v50,fine,PencilHolder\WObj:=PAPER;
MoveL Offs(Target_drawing_origin,-91,157,0),v50,fine,PencilHolder\WObj:=PAPER;
MoveL Offs(Target_drawing_origin,-91,183,0),v50,fine,PencilHolder\WObj:=PAPER;
MoveL Offs(Target_drawing_origin,-91,195,0),v50,fine,PencilHolder\WObj:=PAPER;
MoveL Offs(Target_drawing_origin,-91,216,0),v50,fine,PencilHolder\WObj:=PAPER;
MoveL Offs(Target_drawing_origin,-91,227,0),v50,fine,PencilHolder\WObj:=PAPER;
MoveL Offs(Target_drawing_origin,-91,248,0),v50,fine,PencilHolder\WObj:=PAPER;
MoveL Offs(Target_drawing_origin,-92,43,0),v50,fine,PencilHolder\WObj:=PAPER;
MoveL Offs(Target_drawing_origin,-92,118,0),v50,fine,PencilHolder\WObj:=PAPER;
MoveL Offs(Target_drawing_origin,-92,157,0),v50,fine,PencilHolder\WObj:=PAPER;
MoveL Offs(Target_drawing_origin,-92,183,0),v50,fine,PencilHolder\WObj:=PAPER;
MoveL Offs(Target_drawing_origin,-92,195,0),v50,fine,PencilHolder\WObj:=PAPER;
MoveL Offs(Target_drawing_origin,-92,216,0),v50,fine,PencilHolder\WObj:=PAPER;
MoveL Offs(Target_drawing_origin,-92,227,0),v50,fine,PencilHolder\WObj:=PAPER;
MoveL Offs(Target_drawing_origin,-92,248,0),v50,fine,PencilHolder\WObj:=PAPER;
MoveL Offs(Target_drawing_origin,-93,43,0),v50,fine,PencilHolder\WObj:=PAPER;
MoveL Offs(Target_drawing_origin,-93,118,0),v50,fine,PencilHolder\WObj:=PAPER;
MoveL Offs(Target_drawing_origin,-93,157,0),v50,fine,PencilHolder\WObj:=PAPER;
MoveL Offs(Target_drawing_origin,-93,183,0),v50,fine,PencilHolder\WObj:=PAPER;
MoveL Offs(Target_drawing_origin,-93,195,0),v50,fine,PencilHolder\WObj:=PAPER;
MoveL Offs(Target_drawing_origin,-93,216,0),v50,fine,PencilHolder\WObj:=PAPER;
MoveL Offs(Target_drawing_origin,-93,227,0),v50,fine,PencilHolder\WObj:=PAPER;
MoveL Offs(Target_drawing_origin,-93,248,0),v50,fine,PencilHolder\WObj:=PAPER;
MoveL Offs(Target_drawing_origin,-94,43,0),v50,fine,PencilHolder\WObj:=PAPER;
MoveL Offs(Target_drawing_origin,-94,118,0),v50,fine,PencilHolder\WObj:=PAPER;
MoveL Offs(Target_drawing_origin,-94,157,0),v50,fine,PencilHolder\WObj:=PAPER;
MoveL Offs(Target_drawing_origin,-94,183,0),v50,fine,PencilHolder\WObj:=PAPER;
MoveL Offs(Target_drawing_origin,-94,195,0),v50,fine,PencilHolder\WObj:=PAPER;
MoveL Offs(Target_drawing_origin,-94,216,0),v50,fine,PencilHolder\WObj:=PAPER;
MoveL Offs(Target_drawing_origin,-94,227,0),v50,fine,PencilHolder\WObj:=PAPER;
MoveL Offs(Target_drawing_origin,-94,248,0),v50,fine,PencilHolder\WObj:=PAPER;
MoveL Offs(Target_drawing_origin,-95,43,0),v50,fine,PencilHolder\WObj:=PAPER;
MoveL Offs(Target_drawing_origin,-95,118,0),v50,fine,PencilHolder\WObj:=PAPER;
MoveL Offs(Target_drawing_origin,-95,157,0),v50,fine,PencilHolder\WObj:=PAPER;
MoveL Offs(Target_drawing_origin,-95,183,0),v50,fine,PencilHolder\WObj:=PAPER;
MoveL Offs(Target_drawing_origin,-95,195,0),v50,fine,PencilHolder\WObj:=PAPER;
MoveL Offs(Target_drawing_origin,-95,216,0),v50,fine,PencilHolder\WObj:=PAPER;
MoveL Offs(Target_drawing_origin,-95,227,0),v50,fine,PencilHolder\WObj:=PAPER;
MoveL Offs(Target_drawing_origin,-95,248,0),v50,fine,PencilHolder\WObj:=PAPER;
MoveL Offs(Target_drawing_origin,-96,43,0),v50,fine,PencilHolder\WObj:=PAPER;
MoveL Offs(Target_drawing_origin,-96,118,0),v50,fine,PencilHolder\WObj:=PAPER;
MoveL Offs(Target_drawing_origin,-96,157,0),v50,fine,PencilHolder\WObj:=PAPER;
MoveL Offs(Target_drawing_origin,-96,183,0),v50,fine,PencilHolder\WObj:=PAPER;
MoveL Offs(Target_drawing_origin,-96,195,0),v50,fine,PencilHolder\WObj:=PAPER;
MoveL Offs(Target_drawing_origin,-96,216,0),v50,fine,PencilHolder\WObj:=PAPER;
MoveL Offs(Target_drawing_origin,-96,227,0),v50,fine,PencilHolder\WObj:=PAPER;
MoveL Offs(Target_drawing_origin,-96,248,0),v50,fine,PencilHolder\WObj:=PAPER;
MoveL Offs(Target_drawing_origin,-97,48,0),v50,fine,PencilHolder\WObj:=PAPER;
MoveL Offs(Target_drawing_origin,-97,113,0),v50,fine,PencilHolder\WObj:=PAPER;
MoveL Offs(Target_drawing_origin,-97,157,0),v50,fine,PencilHolder\WObj:=PAPER;
MoveL Offs(Target_drawing_origin,-97,183,0),v50,fine,PencilHolder\WObj:=PAPER;
MoveL Offs(Target_drawing_origin,-97,195,0),v50,fine,PencilHolder\WObj:=PAPER;
MoveL Offs(Target_drawing_origin,-97,216,0),v50,fine,PencilHolder\WObj:=PAPER;
MoveL Offs(Target_drawing_origin,-97,227,0),v50,fine,PencilHolder\WObj:=PAPER;
MoveL Offs(Target_drawing_origin,-97,248,0),v50,fine,PencilHolder\WObj:=PAPER;
MoveL Offs(Target_drawing_origin,-98,49,0),v50,fine,PencilHolder\WObj:=PAPER;
MoveL Offs(Target_drawing_origin,-98,113,0),v50,fine,PencilHolder\WObj:=PAPER;
MoveL Offs(Target_drawing_origin,-98,157,0),v50,fine,PencilHolder\WObj:=PAPER;
MoveL Offs(Target_drawing_origin,-98,183,0),v50,fine,PencilHolder\WObj:=PAPER;
MoveL Offs(Target_drawing_origin,-98,195,0),v50,fine,PencilHolder\WObj:=PAPER;
MoveL Offs(Target_drawing_origin,-98,216,0),v50,fine,PencilHolder\WObj:=PAPER;
MoveL Offs(Target_drawing_origin,-98,227,0),v50,fine,PencilHolder\WObj:=PAPER;
MoveL Offs(Target_drawing_origin,-98,248,0),v50,fine,PencilHolder\WObj:=PAPER;
MoveL Offs(Target_drawing_origin,-99,49,0),v50,fine,PencilHolder\WObj:=PAPER;
MoveL Offs(Target_drawing_origin,-99,113,0),v50,fine,PencilHolder\WObj:=PAPER;
MoveL Offs(Target_drawing_origin,-99,157,0),v50,fine,PencilHolder\WObj:=PAPER;
MoveL Offs(Target_drawing_origin,-99,183,0),v50,fine,PencilHolder\WObj:=PAPER;
MoveL Offs(Target_drawing_origin,-99,195,0),v50,fine,PencilHolder\WObj:=PAPER;
MoveL Offs(Target_drawing_origin,-99,216,0),v50,fine,PencilHolder\WObj:=PAPER;
MoveL Offs(Target_drawing_origin,-99,227,0),v50,fine,PencilHolder\WObj:=PAPER;
MoveL Offs(Target_drawing_origin,-99,248,0),v50,fine,PencilHolder\WObj:=PAPER;
MoveL Offs(Target_drawing_origin,-100,49,0),v50,fine,PencilHolder\WObj:=PAPER;
MoveL Offs(Target_drawing_origin,-100,113,0),v50,fine,PencilHolder\WObj:=PAPER;
MoveL Offs(Target_drawing_origin,-100,157,0),v50,fine,PencilHolder\WObj:=PAPER;
MoveL Offs(Target_drawing_origin,-100,183,0),v50,fine,PencilHolder\WObj:=PAPER;
MoveL Offs(Target_drawing_origin,-100,195,0),v50,fine,PencilHolder\WObj:=PAPER;
MoveL Offs(Target_drawing_origin,-100,216,0),v50,fine,PencilHolder\WObj:=PAPER;
MoveL Offs(Target_drawing_origin,-100,227,0),v50,fine,PencilHolder\WObj:=PAPER;
MoveL Offs(Target_drawing_origin,-100,248,0),v50,fine,PencilHolder\WObj:=PAPER;
MoveL Offs(Target_drawing_origin,-101,49,0),v50,fine,PencilHolder\WObj:=PAPER;
MoveL Offs(Target_drawing_origin,-101,113,0),v50,fine,PencilHolder\WObj:=PAPER;
MoveL Offs(Target_drawing_origin,-101,157,0),v50,fine,PencilHolder\WObj:=PAPER;
MoveL Offs(Target_drawing_origin,-101,183,0),v50,fine,PencilHolder\WObj:=PAPER;
MoveL Offs(Target_drawing_origin,-101,195,0),v50,fine,PencilHolder\WObj:=PAPER;
MoveL Offs(Target_drawing_origin,-101,216,0),v50,fine,PencilHolder\WObj:=PAPER;
MoveL Offs(Target_drawing_origin,-101,227,0),v50,fine,PencilHolder\WObj:=PAPER;
MoveL Offs(Target_drawing_origin,-101,248,0),v50,fine,PencilHolder\WObj:=PAPER;
MoveL Offs(Target_drawing_origin,-102,49,0),v50,fine,PencilHolder\WObj:=PAPER;
MoveL Offs(Target_drawing_origin,-102,113,0),v50,fine,PencilHolder\WObj:=PAPER;
MoveL Offs(Target_drawing_origin,-102,157,0),v50,fine,PencilHolder\WObj:=PAPER;
MoveL Offs(Target_drawing_origin,-102,183,0),v50,fine,PencilHolder\WObj:=PAPER;
MoveL Offs(Target_drawing_origin,-102,195,0),v50,fine,PencilHolder\WObj:=PAPER;
MoveL Offs(Target_drawing_origin,-102,216,0),v50,fine,PencilHolder\WObj:=PAPER;
MoveL Offs(Target_drawing_origin,-102,227,0),v50,fine,PencilHolder\WObj:=PAPER;
MoveL Offs(Target_drawing_origin,-102,248,0),v50,fine,PencilHolder\WObj:=PAPER;
MoveL Offs(Target_drawing_origin,-103,54,0),v50,fine,PencilHolder\WObj:=PAPER;
MoveL Offs(Target_drawing_origin,-103,113,0),v50,fine,PencilHolder\WObj:=PAPER;
MoveL Offs(Target_drawing_origin,-103,157,0),v50,fine,PencilHolder\WObj:=PAPER;
MoveL Offs(Target_drawing_origin,-103,183,0),v50,fine,PencilHolder\WObj:=PAPER;
MoveL Offs(Target_drawing_origin,-103,189,0),v50,fine,PencilHolder\WObj:=PAPER;
MoveL Offs(Target_drawing_origin,-103,216,0),v50,fine,PencilHolder\WObj:=PAPER;
MoveL Offs(Target_drawing_origin,-103,227,0),v50,fine,PencilHolder\WObj:=PAPER;
MoveL Offs(Target_drawing_origin,-103,248,0),v50,fine,PencilHolder\WObj:=PAPER;
MoveL Offs(Target_drawing_origin,-104,54,0),v50,fine,PencilHolder\WObj:=PAPER;
MoveL Offs(Target_drawing_origin,-104,113,0),v50,fine,PencilHolder\WObj:=PAPER;
MoveL Offs(Target_drawing_origin,-104,157,0),v50,fine,PencilHolder\WObj:=PAPER;
MoveL Offs(Target_drawing_origin,-104,183,0),v50,fine,PencilHolder\WObj:=PAPER;
MoveL Offs(Target_drawing_origin,-104,189,0),v50,fine,PencilHolder\WObj:=PAPER;
MoveL Offs(Target_drawing_origin,-104,216,0),v50,fine,PencilHolder\WObj:=PAPER;
MoveL Offs(Target_drawing_origin,-104,227,0),v50,fine,PencilHolder\WObj:=PAPER;
MoveL Offs(Target_drawing_origin,-104,248,0),v50,fine,PencilHolder\WObj:=PAPER;
MoveL Offs(Target_drawing_origin,-105,54,0),v50,fine,PencilHolder\WObj:=PAPER;
MoveL Offs(Target_drawing_origin,-105,113,0),v50,fine,PencilHolder\WObj:=PAPER;
MoveL Offs(Target_drawing_origin,-105,157,0),v50,fine,PencilHolder\WObj:=PAPER;
MoveL Offs(Target_drawing_origin,-105,183,0),v50,fine,PencilHolder\WObj:=PAPER;
MoveL Offs(Target_drawing_origin,-105,189,0),v50,fine,PencilHolder\WObj:=PAPER;
MoveL Offs(Target_drawing_origin,-105,216,0),v50,fine,PencilHolder\WObj:=PAPER;
MoveL Offs(Target_drawing_origin,-105,227,0),v50,fine,PencilHolder\WObj:=PAPER;
MoveL Offs(Target_drawing_origin,-105,248,0),v50,fine,PencilHolder\WObj:=PAPER;
MoveL Offs(Target_drawing_origin,-106,54,0),v50,fine,PencilHolder\WObj:=PAPER;
MoveL Offs(Target_drawing_origin,-106,113,0),v50,fine,PencilHolder\WObj:=PAPER;
MoveL Offs(Target_drawing_origin,-106,157,0),v50,fine,PencilHolder\WObj:=PAPER;
MoveL Offs(Target_drawing_origin,-106,183,0),v50,fine,PencilHolder\WObj:=PAPER;
MoveL Offs(Target_drawing_origin,-106,189,0),v50,fine,PencilHolder\WObj:=PAPER;
MoveL Offs(Target_drawing_origin,-106,216,0),v50,fine,PencilHolder\WObj:=PAPER;
MoveL Offs(Target_drawing_origin,-106,227,0),v50,fine,PencilHolder\WObj:=PAPER;
MoveL Offs(Target_drawing_origin,-106,248,0),v50,fine,PencilHolder\WObj:=PAPER;
MoveL Offs(Target_drawing_origin,-107,54,0),v50,fine,PencilHolder\WObj:=PAPER;
MoveL Offs(Target_drawing_origin,-107,113,0),v50,fine,PencilHolder\WObj:=PAPER;
MoveL Offs(Target_drawing_origin,-107,157,0),v50,fine,PencilHolder\WObj:=PAPER;
MoveL Offs(Target_drawing_origin,-107,183,0),v50,fine,PencilHolder\WObj:=PAPER;
MoveL Offs(Target_drawing_origin,-107,189,0),v50,fine,PencilHolder\WObj:=PAPER;
MoveL Offs(Target_drawing_origin,-107,216,0),v50,fine,PencilHolder\WObj:=PAPER;
MoveL Offs(Target_drawing_origin,-107,227,0),v50,fine,PencilHolder\WObj:=PAPER;
MoveL Offs(Target_drawing_origin,-107,248,0),v50,fine,PencilHolder\WObj:=PAPER;
MoveL Offs(Target_drawing_origin,-108,59,0),v50,fine,PencilHolder\WObj:=PAPER;
MoveL Offs(Target_drawing_origin,-108,108,0),v50,fine,PencilHolder\WObj:=PAPER;
MoveL Offs(Target_drawing_origin,-108,152,0),v50,fine,PencilHolder\WObj:=PAPER;
MoveL Offs(Target_drawing_origin,-108,183,0),v50,fine,PencilHolder\WObj:=PAPER;
MoveL Offs(Target_drawing_origin,-108,189,0),v50,fine,PencilHolder\WObj:=PAPER;
MoveL Offs(Target_drawing_origin,-108,216,0),v50,fine,PencilHolder\WObj:=PAPER;
MoveL Offs(Target_drawing_origin,-108,227,0),v50,fine,PencilHolder\WObj:=PAPER;
MoveL Offs(Target_drawing_origin,-108,248,0),v50,fine,PencilHolder\WObj:=PAPER;
MoveL Offs(Target_drawing_origin,-109,59,0),v50,fine,PencilHolder\WObj:=PAPER;
MoveL Offs(Target_drawing_origin,-109,107,0),v50,fine,PencilHolder\WObj:=PAPER;
MoveL Offs(Target_drawing_origin,-109,152,0),v50,fine,PencilHolder\WObj:=PAPER;
MoveL Offs(Target_drawing_origin,-109,183,0),v50,fine,PencilHolder\WObj:=PAPER;
MoveL Offs(Target_drawing_origin,-109,189,0),v50,fine,PencilHolder\WObj:=PAPER;
MoveL Offs(Target_drawing_origin,-109,216,0),v50,fine,PencilHolder\WObj:=PAPER;
MoveL Offs(Target_drawing_origin,-109,227,0),v50,fine,PencilHolder\WObj:=PAPER;
MoveL Offs(Target_drawing_origin,-109,248,0),v50,fine,PencilHolder\WObj:=PAPER;
MoveL Offs(Target_drawing_origin,-110,59,0),v50,fine,PencilHolder\WObj:=PAPER;
MoveL Offs(Target_drawing_origin,-110,107,0),v50,fine,PencilHolder\WObj:=PAPER;
MoveL Offs(Target_drawing_origin,-110,152,0),v50,fine,PencilHolder\WObj:=PAPER;
MoveL Offs(Target_drawing_origin,-110,183,0),v50,fine,PencilHolder\WObj:=PAPER;
MoveL Offs(Target_drawing_origin,-110,189,0),v50,fine,PencilHolder\WObj:=PAPER;
MoveL Offs(Target_drawing_origin,-110,216,0),v50,fine,PencilHolder\WObj:=PAPER;
MoveL Offs(Target_drawing_origin,-110,227,0),v50,fine,PencilHolder\WObj:=PAPER;
MoveL Offs(Target_drawing_origin,-110,248,0),v50,fine,PencilHolder\WObj:=PAPER;
MoveL Offs(Target_drawing_origin,-111,59,0),v50,fine,PencilHolder\WObj:=PAPER;
MoveL Offs(Target_drawing_origin,-111,107,0),v50,fine,PencilHolder\WObj:=PAPER;
MoveL Offs(Target_drawing_origin,-111,152,0),v50,fine,PencilHolder\WObj:=PAPER;
MoveL Offs(Target_drawing_origin,-111,183,0),v50,fine,PencilHolder\WObj:=PAPER;
MoveL Offs(Target_drawing_origin,-111,189,0),v50,fine,PencilHolder\WObj:=PAPER;
MoveL Offs(Target_drawing_origin,-111,216,0),v50,fine,PencilHolder\WObj:=PAPER;
MoveL Offs(Target_drawing_origin,-111,227,0),v50,fine,PencilHolder\WObj:=PAPER;
MoveL Offs(Target_drawing_origin,-111,248,0),v50,fine,PencilHolder\WObj:=PAPER;
MoveL Offs(Target_drawing_origin,-112,59,0),v50,fine,PencilHolder\WObj:=PAPER;
MoveL Offs(Target_drawing_origin,-112,107,0),v50,fine,PencilHolder\WObj:=PAPER;
MoveL Offs(Target_drawing_origin,-112,152,0),v50,fine,PencilHolder\WObj:=PAPER;
MoveL Offs(Target_drawing_origin,-112,183,0),v50,fine,PencilHolder\WObj:=PAPER;
MoveL Offs(Target_drawing_origin,-112,189,0),v50,fine,PencilHolder\WObj:=PAPER;
MoveL Offs(Target_drawing_origin,-112,216,0),v50,fine,PencilHolder\WObj:=PAPER;
MoveL Offs(Target_drawing_origin,-112,227,0),v50,fine,PencilHolder\WObj:=PAPER;
MoveL Offs(Target_drawing_origin,-112,248,0),v50,fine,PencilHolder\WObj:=PAPER;
MoveL Offs(Target_drawing_origin,-113,60,0),v50,fine,PencilHolder\WObj:=PAPER;
MoveL Offs(Target_drawing_origin,-113,107,0),v50,fine,PencilHolder\WObj:=PAPER;
MoveL Offs(Target_drawing_origin,-113,152,0),v50,fine,PencilHolder\WObj:=PAPER;
MoveL Offs(Target_drawing_origin,-113,183,0),v50,fine,PencilHolder\WObj:=PAPER;
MoveL Offs(Target_drawing_origin,-113,189,0),v50,fine,PencilHolder\WObj:=PAPER;
MoveL Offs(Target_drawing_origin,-113,216,0),v50,fine,PencilHolder\WObj:=PAPER;
MoveL Offs(Target_drawing_origin,-113,227,0),v50,fine,PencilHolder\WObj:=PAPER;
MoveL Offs(Target_drawing_origin,-113,248,0),v50,fine,PencilHolder\WObj:=PAPER;
MoveL Offs(Target_drawing_origin,-114,66,0),v50,fine,PencilHolder\WObj:=PAPER;
MoveL Offs(Target_drawing_origin,-114,102,0),v50,fine,PencilHolder\WObj:=PAPER;
MoveL Offs(Target_drawing_origin,-114,152,0),v50,fine,PencilHolder\WObj:=PAPER;
MoveL Offs(Target_drawing_origin,-114,183,0),v50,fine,PencilHolder\WObj:=PAPER;
MoveL Offs(Target_drawing_origin,-114,189,0),v50,fine,PencilHolder\WObj:=PAPER;
MoveL Offs(Target_drawing_origin,-114,216,0),v50,fine,PencilHolder\WObj:=PAPER;
MoveL Offs(Target_drawing_origin,-114,227,0),v50,fine,PencilHolder\WObj:=PAPER;
MoveL Offs(Target_drawing_origin,-114,248,0),v50,fine,PencilHolder\WObj:=PAPER;
MoveL Offs(Target_drawing_origin,-115,66,0),v50,fine,PencilHolder\WObj:=PAPER;
MoveL Offs(Target_drawing_origin,-115,102,0),v50,fine,PencilHolder\WObj:=PAPER;
MoveL Offs(Target_drawing_origin,-115,152,0),v50,fine,PencilHolder\WObj:=PAPER;
MoveL Offs(Target_drawing_origin,-115,183,0),v50,fine,PencilHolder\WObj:=PAPER;
MoveL Offs(Target_drawing_origin,-115,189,0),v50,fine,PencilHolder\WObj:=PAPER;
MoveL Offs(Target_drawing_origin,-115,216,0),v50,fine,PencilHolder\WObj:=PAPER;
MoveL Offs(Target_drawing_origin,-115,227,0),v50,fine,PencilHolder\WObj:=PAPER;
MoveL Offs(Target_drawing_origin,-115,248,0),v50,fine,PencilHolder\WObj:=PAPER;
MoveL Offs(Target_drawing_origin,-116,66,0),v50,fine,PencilHolder\WObj:=PAPER;
MoveL Offs(Target_drawing_origin,-116,102,0),v50,fine,PencilHolder\WObj:=PAPER;
MoveL Offs(Target_drawing_origin,-116,152,0),v50,fine,PencilHolder\WObj:=PAPER;
MoveL Offs(Target_drawing_origin,-116,183,0),v50,fine,PencilHolder\WObj:=PAPER;
MoveL Offs(Target_drawing_origin,-116,189,0),v50,fine,PencilHolder\WObj:=PAPER;
MoveL Offs(Target_drawing_origin,-116,216,0),v50,fine,PencilHolder\WObj:=PAPER;
MoveL Offs(Target_drawing_origin,-116,227,0),v50,fine,PencilHolder\WObj:=PAPER;
MoveL Offs(Target_drawing_origin,-116,248,0),v50,fine,PencilHolder\WObj:=PAPER;
MoveL Offs(Target_drawing_origin,-117,66,0),v50,fine,PencilHolder\WObj:=PAPER;
MoveL Offs(Target_drawing_origin,-117,102,0),v50,fine,PencilHolder\WObj:=PAPER;
MoveL Offs(Target_drawing_origin,-117,152,0),v50,fine,PencilHolder\WObj:=PAPER;
MoveL Offs(Target_drawing_origin,-117,183,0),v50,fine,PencilHolder\WObj:=PAPER;
MoveL Offs(Target_drawing_origin,-117,189,0),v50,fine,PencilHolder\WObj:=PAPER;
MoveL Offs(Target_drawing_origin,-117,216,0),v50,fine,PencilHolder\WObj:=PAPER;
MoveL Offs(Target_drawing_origin,-117,227,0),v50,fine,PencilHolder\WObj:=PAPER;
MoveL Offs(Target_drawing_origin,-117,248,0),v50,fine,PencilHolder\WObj:=PAPER;
MoveL Offs(Target_drawing_origin,-118,66,0),v50,fine,PencilHolder\WObj:=PAPER;
MoveL Offs(Target_drawing_origin,-118,102,0),v50,fine,PencilHolder\WObj:=PAPER;
MoveL Offs(Target_drawing_origin,-118,152,0),v50,fine,PencilHolder\WObj:=PAPER;
MoveL Offs(Target_drawing_origin,-118,183,0),v50,fine,PencilHolder\WObj:=PAPER;
MoveL Offs(Target_drawing_origin,-118,189,0),v50,fine,PencilHolder\WObj:=PAPER;
MoveL Offs(Target_drawing_origin,-118,216,0),v50,fine,PencilHolder\WObj:=PAPER;
MoveL Offs(Target_drawing_origin,-118,227,0),v50,fine,PencilHolder\WObj:=PAPER;
MoveL Offs(Target_drawing_origin,-118,248,0),v50,fine,PencilHolder\WObj:=PAPER;
MoveL Offs(Target_drawing_origin,-119,70,0),v50,fine,PencilHolder\WObj:=PAPER;
MoveL Offs(Target_drawing_origin,-119,97,0),v50,fine,PencilHolder\WObj:=PAPER;
MoveL Offs(Target_drawing_origin,-119,152,0),v50,fine,PencilHolder\WObj:=PAPER;
MoveL Offs(Target_drawing_origin,-119,178,0),v50,fine,PencilHolder\WObj:=PAPER;
MoveL Offs(Target_drawing_origin,-119,184,0),v50,fine,PencilHolder\WObj:=PAPER;
MoveL Offs(Target_drawing_origin,-119,216,0),v50,fine,PencilHolder\WObj:=PAPER;
MoveL Offs(Target_drawing_origin,-119,227,0),v50,fine,PencilHolder\WObj:=PAPER;
MoveL Offs(Target_drawing_origin,-119,248,0),v50,fine,PencilHolder\WObj:=PAPER;
MoveL Offs(Target_drawing_origin,-120,70,0),v50,fine,PencilHolder\WObj:=PAPER;
MoveL Offs(Target_drawing_origin,-120,97,0),v50,fine,PencilHolder\WObj:=PAPER;
MoveL Offs(Target_drawing_origin,-120,152,0),v50,fine,PencilHolder\WObj:=PAPER;
MoveL Offs(Target_drawing_origin,-120,178,0),v50,fine,PencilHolder\WObj:=PAPER;
MoveL Offs(Target_drawing_origin,-120,184,0),v50,fine,PencilHolder\WObj:=PAPER;
MoveL Offs(Target_drawing_origin,-120,216,0),v50,fine,PencilHolder\WObj:=PAPER;
MoveL Offs(Target_drawing_origin,-120,227,0),v50,fine,PencilHolder\WObj:=PAPER;
MoveL Offs(Target_drawing_origin,-120,248,0),v50,fine,PencilHolder\WObj:=PAPER;
MoveL Offs(Target_drawing_origin,-121,70,0),v50,fine,PencilHolder\WObj:=PAPER;
MoveL Offs(Target_drawing_origin,-121,97,0),v50,fine,PencilHolder\WObj:=PAPER;
MoveL Offs(Target_drawing_origin,-121,152,0),v50,fine,PencilHolder\WObj:=PAPER;
MoveL Offs(Target_drawing_origin,-121,178,0),v50,fine,PencilHolder\WObj:=PAPER;
MoveL Offs(Target_drawing_origin,-121,184,0),v50,fine,PencilHolder\WObj:=PAPER;
MoveL Offs(Target_drawing_origin,-121,216,0),v50,fine,PencilHolder\WObj:=PAPER;
MoveL Offs(Target_drawing_origin,-121,227,0),v50,fine,PencilHolder\WObj:=PAPER;
MoveL Offs(Target_drawing_origin,-121,248,0),v50,fine,PencilHolder\WObj:=PAPER;
MoveL Offs(Target_drawing_origin,-122,70,0),v50,fine,PencilHolder\WObj:=PAPER;
MoveL Offs(Target_drawing_origin,-122,97,0),v50,fine,PencilHolder\WObj:=PAPER;
MoveL Offs(Target_drawing_origin,-122,152,0),v50,fine,PencilHolder\WObj:=PAPER;
MoveL Offs(Target_drawing_origin,-122,178,0),v50,fine,PencilHolder\WObj:=PAPER;
MoveL Offs(Target_drawing_origin,-122,184,0),v50,fine,PencilHolder\WObj:=PAPER;
MoveL Offs(Target_drawing_origin,-122,216,0),v50,fine,PencilHolder\WObj:=PAPER;
MoveL Offs(Target_drawing_origin,-122,227,0),v50,fine,PencilHolder\WObj:=PAPER;
MoveL Offs(Target_drawing_origin,-122,248,0),v50,fine,PencilHolder\WObj:=PAPER;
MoveL Offs(Target_drawing_origin,-123,70,0),v50,fine,PencilHolder\WObj:=PAPER;
MoveL Offs(Target_drawing_origin,-123,97,0),v50,fine,PencilHolder\WObj:=PAPER;
MoveL Offs(Target_drawing_origin,-123,152,0),v50,fine,PencilHolder\WObj:=PAPER;
MoveL Offs(Target_drawing_origin,-123,178,0),v50,fine,PencilHolder\WObj:=PAPER;
MoveL Offs(Target_drawing_origin,-123,184,0),v50,fine,PencilHolder\WObj:=PAPER;
MoveL Offs(Target_drawing_origin,-123,216,0),v50,fine,PencilHolder\WObj:=PAPER;
MoveL Offs(Target_drawing_origin,-123,227,0),v50,fine,PencilHolder\WObj:=PAPER;
MoveL Offs(Target_drawing_origin,-123,248,0),v50,fine,PencilHolder\WObj:=PAPER;
MoveL Offs(Target_drawing_origin,-124,152,0),v50,fine,PencilHolder\WObj:=PAPER;
MoveL Offs(Target_drawing_origin,-124,173,0),v50,fine,PencilHolder\WObj:=PAPER;
MoveL Offs(Target_drawing_origin,-124,184,0),v50,fine,PencilHolder\WObj:=PAPER;
MoveL Offs(Target_drawing_origin,-124,211,0),v50,fine,PencilHolder\WObj:=PAPER;
MoveL Offs(Target_drawing_origin,-124,227,0),v50,fine,PencilHolder\WObj:=PAPER;
MoveL Offs(Target_drawing_origin,-124,253,0),v50,fine,PencilHolder\WObj:=PAPER;
MoveL Offs(Target_drawing_origin,-125,152,0),v50,fine,PencilHolder\WObj:=PAPER;
MoveL Offs(Target_drawing_origin,-125,172,0),v50,fine,PencilHolder\WObj:=PAPER;
MoveL Offs(Target_drawing_origin,-125,184,0),v50,fine,PencilHolder\WObj:=PAPER;
MoveL Offs(Target_drawing_origin,-125,210,0),v50,fine,PencilHolder\WObj:=PAPER;
MoveL Offs(Target_drawing_origin,-125,227,0),v50,fine,PencilHolder\WObj:=PAPER;
MoveL Offs(Target_drawing_origin,-125,254,0),v50,fine,PencilHolder\WObj:=PAPER;
MoveL Offs(Target_drawing_origin,-126,152,0),v50,fine,PencilHolder\WObj:=PAPER;
MoveL Offs(Target_drawing_origin,-126,172,0),v50,fine,PencilHolder\WObj:=PAPER;
MoveL Offs(Target_drawing_origin,-126,184,0),v50,fine,PencilHolder\WObj:=PAPER;
MoveL Offs(Target_drawing_origin,-126,210,0),v50,fine,PencilHolder\WObj:=PAPER;
MoveL Offs(Target_drawing_origin,-126,227,0),v50,fine,PencilHolder\WObj:=PAPER;
MoveL Offs(Target_drawing_origin,-126,254,0),v50,fine,PencilHolder\WObj:=PAPER;
MoveL Offs(Target_drawing_origin,-127,152,0),v50,fine,PencilHolder\WObj:=PAPER;
MoveL Offs(Target_drawing_origin,-127,172,0),v50,fine,PencilHolder\WObj:=PAPER;
MoveL Offs(Target_drawing_origin,-127,184,0),v50,fine,PencilHolder\WObj:=PAPER;
MoveL Offs(Target_drawing_origin,-127,210,0),v50,fine,PencilHolder\WObj:=PAPER;
MoveL Offs(Target_drawing_origin,-127,227,0),v50,fine,PencilHolder\WObj:=PAPER;
MoveL Offs(Target_drawing_origin,-127,254,0),v50,fine,PencilHolder\WObj:=PAPER;
MoveL Offs(Target_drawing_origin,-128,152,0),v50,fine,PencilHolder\WObj:=PAPER;
MoveL Offs(Target_drawing_origin,-128,172,0),v50,fine,PencilHolder\WObj:=PAPER;
MoveL Offs(Target_drawing_origin,-128,184,0),v50,fine,PencilHolder\WObj:=PAPER;
MoveL Offs(Target_drawing_origin,-128,210,0),v50,fine,PencilHolder\WObj:=PAPER;
MoveL Offs(Target_drawing_origin,-128,227,0),v50,fine,PencilHolder\WObj:=PAPER;
MoveL Offs(Target_drawing_origin,-128,254,0),v50,fine,PencilHolder\WObj:=PAPER;
MoveL Offs(Target_drawing_origin,-129,152,0),v50,fine,PencilHolder\WObj:=PAPER;
MoveL Offs(Target_drawing_origin,-129,173,0),v50,fine,PencilHolder\WObj:=PAPER;
MoveL Offs(Target_drawing_origin,-129,184,0),v50,fine,PencilHolder\WObj:=PAPER;
MoveL Offs(Target_drawing_origin,-129,210,0),v50,fine,PencilHolder\WObj:=PAPER;
MoveL Offs(Target_drawing_origin,-129,227,0),v50,fine,PencilHolder\WObj:=PAPER;
MoveL Offs(Target_drawing_origin,-129,254,0),v50,fine,PencilHolder\WObj:=PAPER;
MoveL Offs(Target_drawing_origin,-130,152,0),v50,fine,PencilHolder\WObj:=PAPER;
MoveL Offs(Target_drawing_origin,-130,210,0),v50,fine,PencilHolder\WObj:=PAPER;
MoveL Offs(Target_drawing_origin,-130,227,0),v50,fine,PencilHolder\WObj:=PAPER;
MoveL Offs(Target_drawing_origin,-130,254,0),v50,fine,PencilHolder\WObj:=PAPER;
MoveL Offs(Target_drawing_origin,-131,152,0),v50,fine,PencilHolder\WObj:=PAPER;
MoveL Offs(Target_drawing_origin,-131,210,0),v50,fine,PencilHolder\WObj:=PAPER;
MoveL Offs(Target_drawing_origin,-131,227,0),v50,fine,PencilHolder\WObj:=PAPER;
MoveL Offs(Target_drawing_origin,-131,254,0),v50,fine,PencilHolder\WObj:=PAPER;
MoveL Offs(Target_drawing_origin,-132,152,0),v50,fine,PencilHolder\WObj:=PAPER;
MoveL Offs(Target_drawing_origin,-132,210,0),v50,fine,PencilHolder\WObj:=PAPER;
MoveL Offs(Target_drawing_origin,-132,227,0),v50,fine,PencilHolder\WObj:=PAPER;
MoveL Offs(Target_drawing_origin,-132,254,0),v50,fine,PencilHolder\WObj:=PAPER;
MoveL Offs(Target_drawing_origin,-133,152,0),v50,fine,PencilHolder\WObj:=PAPER;
MoveL Offs(Target_drawing_origin,-133,210,0),v50,fine,PencilHolder\WObj:=PAPER;
MoveL Offs(Target_drawing_origin,-133,227,0),v50,fine,PencilHolder\WObj:=PAPER;
MoveL Offs(Target_drawing_origin,-133,254,0),v50,fine,PencilHolder\WObj:=PAPER;
MoveL Offs(Target_drawing_origin,-134,152,0),v50,fine,PencilHolder\WObj:=PAPER;
MoveL Offs(Target_drawing_origin,-134,210,0),v50,fine,PencilHolder\WObj:=PAPER;
MoveL Offs(Target_drawing_origin,-134,227,0),v50,fine,PencilHolder\WObj:=PAPER;
MoveL Offs(Target_drawing_origin,-134,254,0),v50,fine,PencilHolder\WObj:=PAPER;
MoveL Offs(Target_drawing_origin,-135,152,0),v50,fine,PencilHolder\WObj:=PAPER;
MoveL Offs(Target_drawing_origin,-135,210,0),v50,fine,PencilHolder\WObj:=PAPER;
MoveL Offs(Target_drawing_origin,-135,227,0),v50,fine,PencilHolder\WObj:=PAPER;
MoveL Offs(Target_drawing_origin,-135,254,0),v50,fine,PencilHolder\WObj:=PAPER;
MoveL Offs(Target_drawing_origin,-136,152,0),v50,fine,PencilHolder\WObj:=PAPER;
MoveL Offs(Target_drawing_origin,-136,210,0),v50,fine,PencilHolder\WObj:=PAPER;
MoveL Offs(Target_drawing_origin,-136,227,0),v50,fine,PencilHolder\WObj:=PAPER;
MoveL Offs(Target_drawing_origin,-136,254,0),v50,fine,PencilHolder\WObj:=PAPER;
MoveL Offs(Target_drawing_origin,-137,152,0),v50,fine,PencilHolder\WObj:=PAPER;
MoveL Offs(Target_drawing_origin,-137,210,0),v50,fine,PencilHolder\WObj:=PAPER;
MoveL Offs(Target_drawing_origin,-137,227,0),v50,fine,PencilHolder\WObj:=PAPER;
MoveL Offs(Target_drawing_origin,-137,254,0),v50,fine,PencilHolder\WObj:=PAPER;
MoveL Offs(Target_drawing_origin,-138,152,0),v50,fine,PencilHolder\WObj:=PAPER;
MoveL Offs(Target_drawing_origin,-138,210,0),v50,fine,PencilHolder\WObj:=PAPER;
MoveL Offs(Target_drawing_origin,-138,227,0),v50,fine,PencilHolder\WObj:=PAPER;
MoveL Offs(Target_drawing_origin,-138,254,0),v50,fine,PencilHolder\WObj:=PAPER;
MoveL Offs(Target_drawing_origin,-139,152,0),v50,fine,PencilHolder\WObj:=PAPER;
MoveL Offs(Target_drawing_origin,-139,210,0),v50,fine,PencilHolder\WObj:=PAPER;
MoveL Offs(Target_drawing_origin,-139,227,0),v50,fine,PencilHolder\WObj:=PAPER;
MoveL Offs(Target_drawing_origin,-139,254,0),v50,fine,PencilHolder\WObj:=PAPER;
MoveL Offs(Target_drawing_origin,-140,152,0),v50,fine,PencilHolder\WObj:=PAPER;
MoveL Offs(Target_drawing_origin,-140,210,0),v50,fine,PencilHolder\WObj:=PAPER;
MoveL Offs(Target_drawing_origin,-140,228,0),v50,fine,PencilHolder\WObj:=PAPER;
MoveL Offs(Target_drawing_origin,-140,254,0),v50,fine,PencilHolder\WObj:=PAPER;
MoveL Offs(Target_drawing_origin,-141,152,0),v50,fine,PencilHolder\WObj:=PAPER;
MoveL Offs(Target_drawing_origin,-141,205,0),v50,fine,PencilHolder\WObj:=PAPER;
MoveL Offs(Target_drawing_origin,-141,233,0),v50,fine,PencilHolder\WObj:=PAPER;
MoveL Offs(Target_drawing_origin,-141,254,0),v50,fine,PencilHolder\WObj:=PAPER;
MoveL Offs(Target_drawing_origin,-142,152,0),v50,fine,PencilHolder\WObj:=PAPER;
MoveL Offs(Target_drawing_origin,-142,205,0),v50,fine,PencilHolder\WObj:=PAPER;
MoveL Offs(Target_drawing_origin,-142,233,0),v50,fine,PencilHolder\WObj:=PAPER;
MoveL Offs(Target_drawing_origin,-142,254,0),v50,fine,PencilHolder\WObj:=PAPER;
MoveL Offs(Target_drawing_origin,-143,152,0),v50,fine,PencilHolder\WObj:=PAPER;
MoveL Offs(Target_drawing_origin,-143,205,0),v50,fine,PencilHolder\WObj:=PAPER;
MoveL Offs(Target_drawing_origin,-143,233,0),v50,fine,PencilHolder\WObj:=PAPER;
MoveL Offs(Target_drawing_origin,-143,254,0),v50,fine,PencilHolder\WObj:=PAPER;
MoveL Offs(Target_drawing_origin,-144,152,0),v50,fine,PencilHolder\WObj:=PAPER;
MoveL Offs(Target_drawing_origin,-144,205,0),v50,fine,PencilHolder\WObj:=PAPER;
MoveL Offs(Target_drawing_origin,-144,233,0),v50,fine,PencilHolder\WObj:=PAPER;
MoveL Offs(Target_drawing_origin,-144,254,0),v50,fine,PencilHolder\WObj:=PAPER;
MoveL Offs(Target_drawing_origin,-145,152,0),v50,fine,PencilHolder\WObj:=PAPER;
MoveL Offs(Target_drawing_origin,-145,205,0),v50,fine,PencilHolder\WObj:=PAPER;
MoveL Offs(Target_drawing_origin,-145,233,0),v50,fine,PencilHolder\WObj:=PAPER;
MoveL Offs(Target_drawing_origin,-145,254,0),v50,fine,PencilHolder\WObj:=PAPER;
MoveL Offs(Target_drawing_origin,-146,157,0),v50,fine,PencilHolder\WObj:=PAPER;
MoveL Offs(Target_drawing_origin,-146,200,0),v50,fine,PencilHolder\WObj:=PAPER;
MoveL Offs(Target_drawing_origin,-146,233,0),v50,fine,PencilHolder\WObj:=PAPER;
MoveL Offs(Target_drawing_origin,-146,259,0),v50,fine,PencilHolder\WObj:=PAPER;
MoveL Offs(Target_drawing_origin,-147,157,0),v50,fine,PencilHolder\WObj:=PAPER;
MoveL Offs(Target_drawing_origin,-147,200,0),v50,fine,PencilHolder\WObj:=PAPER;
MoveL Offs(Target_drawing_origin,-147,233,0),v50,fine,PencilHolder\WObj:=PAPER;
MoveL Offs(Target_drawing_origin,-147,259,0),v50,fine,PencilHolder\WObj:=PAPER;
MoveL Offs(Target_drawing_origin,-148,157,0),v50,fine,PencilHolder\WObj:=PAPER;
MoveL Offs(Target_drawing_origin,-148,200,0),v50,fine,PencilHolder\WObj:=PAPER;
MoveL Offs(Target_drawing_origin,-148,233,0),v50,fine,PencilHolder\WObj:=PAPER;
MoveL Offs(Target_drawing_origin,-148,259,0),v50,fine,PencilHolder\WObj:=PAPER;
MoveL Offs(Target_drawing_origin,-149,157,0),v50,fine,PencilHolder\WObj:=PAPER;
MoveL Offs(Target_drawing_origin,-149,200,0),v50,fine,PencilHolder\WObj:=PAPER;
MoveL Offs(Target_drawing_origin,-149,233,0),v50,fine,PencilHolder\WObj:=PAPER;
MoveL Offs(Target_drawing_origin,-149,259,0),v50,fine,PencilHolder\WObj:=PAPER;
MoveL Offs(Target_drawing_origin,-150,157,0),v50,fine,PencilHolder\WObj:=PAPER;
MoveL Offs(Target_drawing_origin,-150,200,0),v50,fine,PencilHolder\WObj:=PAPER;
MoveL Offs(Target_drawing_origin,-150,233,0),v50,fine,PencilHolder\WObj:=PAPER;
MoveL Offs(Target_drawing_origin,-150,259,0),v50,fine,PencilHolder\WObj:=PAPER;
MoveL Offs(Target_drawing_origin,-151,162,0),v50,fine,PencilHolder\WObj:=PAPER;
MoveL Offs(Target_drawing_origin,-151,194,0),v50,fine,PencilHolder\WObj:=PAPER;
MoveL Offs(Target_drawing_origin,-151,233,0),v50,fine,PencilHolder\WObj:=PAPER;
MoveL Offs(Target_drawing_origin,-151,259,0),v50,fine,PencilHolder\WObj:=PAPER;
MoveL Offs(Target_drawing_origin,-152,162,0),v50,fine,PencilHolder\WObj:=PAPER;
MoveL Offs(Target_drawing_origin,-152,194,0),v50,fine,PencilHolder\WObj:=PAPER;
MoveL Offs(Target_drawing_origin,-152,233,0),v50,fine,PencilHolder\WObj:=PAPER;
MoveL Offs(Target_drawing_origin,-152,259,0),v50,fine,PencilHolder\WObj:=PAPER;
MoveL Offs(Target_drawing_origin,-153,162,0),v50,fine,PencilHolder\WObj:=PAPER;
MoveL Offs(Target_drawing_origin,-153,194,0),v50,fine,PencilHolder\WObj:=PAPER;
MoveL Offs(Target_drawing_origin,-153,233,0),v50,fine,PencilHolder\WObj:=PAPER;
MoveL Offs(Target_drawing_origin,-153,259,0),v50,fine,PencilHolder\WObj:=PAPER;
MoveL Offs(Target_drawing_origin,-154,162,0),v50,fine,PencilHolder\WObj:=PAPER;
MoveL Offs(Target_drawing_origin,-154,194,0),v50,fine,PencilHolder\WObj:=PAPER;
MoveL Offs(Target_drawing_origin,-154,233,0),v50,fine,PencilHolder\WObj:=PAPER;
MoveL Offs(Target_drawing_origin,-154,259,0),v50,fine,PencilHolder\WObj:=PAPER;
MoveL Offs(Target_drawing_origin,-155,162,0),v50,fine,PencilHolder\WObj:=PAPER;
MoveL Offs(Target_drawing_origin,-155,194,0),v50,fine,PencilHolder\WObj:=PAPER;
MoveL Offs(Target_drawing_origin,-155,233,0),v50,fine,PencilHolder\WObj:=PAPER;
MoveL Offs(Target_drawing_origin,-155,259,0),v50,fine,PencilHolder\WObj:=PAPER;
MoveL Offs(Target_drawing_origin,-156,163,0),v50,fine,PencilHolder\WObj:=PAPER;
MoveL Offs(Target_drawing_origin,-156,194,0),v50,fine,PencilHolder\WObj:=PAPER;
MoveL Offs(Target_drawing_origin,-156,233,0),v50,fine,PencilHolder\WObj:=PAPER;
MoveL Offs(Target_drawing_origin,-156,259,0),v50,fine,PencilHolder\WObj:=PAPER;
MoveL Offs(Target_drawing_origin,-157,233,0),v50,fine,PencilHolder\WObj:=PAPER;
MoveL Offs(Target_drawing_origin,-157,259,0),v50,fine,PencilHolder\WObj:=PAPER;
MoveL Offs(Target_drawing_origin,-158,233,0),v50,fine,PencilHolder\WObj:=PAPER;
MoveL Offs(Target_drawing_origin,-158,259,0),v50,fine,PencilHolder\WObj:=PAPER;
MoveL Offs(Target_drawing_origin,-159,233,0),v50,fine,PencilHolder\WObj:=PAPER;
MoveL Offs(Target_drawing_origin,-159,259,0),v50,fine,PencilHolder\WObj:=PAPER;
MoveL Offs(Target_drawing_origin,-160,233,0),v50,fine,PencilHolder\WObj:=PAPER;
MoveL Offs(Target_drawing_origin,-160,259,0),v50,fine,PencilHolder\WObj:=PAPER;
MoveL Offs(Target_drawing_origin,-161,233,0),v50,fine,PencilHolder\WObj:=PAPER;
MoveL Offs(Target_drawing_origin,-161,259,0),v50,fine,PencilHolder\WObj:=PAPER;
MoveL Offs(Target_drawing_origin,-162,238,0),v50,fine,PencilHolder\WObj:=PAPER;
MoveL Offs(Target_drawing_origin,-162,259,0),v50,fine,PencilHolder\WObj:=PAPER;
MoveL Offs(Target_drawing_origin,-163,238,0),v50,fine,PencilHolder\WObj:=PAPER;
MoveL Offs(Target_drawing_origin,-163,259,0),v50,fine,PencilHolder\WObj:=PAPER;
MoveL Offs(Target_drawing_origin,-164,238,0),v50,fine,PencilHolder\WObj:=PAPER;
MoveL Offs(Target_drawing_origin,-164,259,0),v50,fine,PencilHolder\WObj:=PAPER;
MoveL Offs(Target_drawing_origin,-165,238,0),v50,fine,PencilHolder\WObj:=PAPER;
MoveL Offs(Target_drawing_origin,-165,259,0),v50,fine,PencilHolder\WObj:=PAPER;
MoveL Offs(Target_drawing_origin,-166,238,0),v50,fine,PencilHolder\WObj:=PAPER;
MoveL Offs(Target_drawing_origin,-166,259,0),v50,fine,PencilHolder\WObj:=PAPER;
MoveL Offs(Target_drawing_origin,-167,238,0),v50,fine,PencilHolder\WObj:=PAPER;
MoveL Offs(Target_drawing_origin,-167,259,0),v50,fine,PencilHolder\WObj:=PAPER;
MoveL Offs(Target_drawing_origin,-168,238,0),v50,fine,PencilHolder\WObj:=PAPER;
MoveL Offs(Target_drawing_origin,-168,259,0),v50,fine,PencilHolder\WObj:=PAPER;
MoveL Offs(Target_drawing_origin,-169,238,0),v50,fine,PencilHolder\WObj:=PAPER;
MoveL Offs(Target_drawing_origin,-169,259,0),v50,fine,PencilHolder\WObj:=PAPER;
MoveL Offs(Target_drawing_origin,-170,238,0),v50,fine,PencilHolder\WObj:=PAPER;
MoveL Offs(Target_drawing_origin,-170,259,0),v50,fine,PencilHolder\WObj:=PAPER;
MoveL Offs(Target_drawing_origin,-171,238,0),v50,fine,PencilHolder\WObj:=PAPER;
MoveL Offs(Target_drawing_origin,-171,259,0),v50,fine,PencilHolder\WObj:=PAPER;
MoveL Offs(Target_drawing_origin,-172,238,0),v50,fine,PencilHolder\WObj:=PAPER;
MoveL Offs(Target_drawing_origin,-172,259,0),v50,fine,PencilHolder\WObj:=PAPER;


